(* CODESYS project l2sivacuumv1.3.3.library
   Company: SLAC - LCLS
   DefaultNamespace: LCLS_Vacuum
   Title: LCLS Vacuum
   Placeholder: LCLS Vacuum
   Author: LCLS ECS-Platforms
   Version: 1.3.3

Project tree, tasks and I/O mapping:
  libraries: LCLS General, * (SLAC); LCLSVacuumSerialDriverLib, 0.0.0 (SLAC - LCLS); PMPS, 0.12.0 (SLAC - LCLS); Tc2_DataExchange, * (Beckhoff Automation GmbH); Tc2_EtherCAT, * (Beckhoff Automation GmbH); Tc2_ModbusSrv, * (Beckhoff Automation GmbH); Tc2_Standard, * (Beckhoff Automation GmbH); Tc2_System, * (Beckhoff Automation GmbH); Tc2_TcpIp, * (Beckhoff Automation GmbH); Tc2_Utilities, * (Beckhoff Automation GmbH); Tc3_EventLogger, * (Beckhoff Automation GmbH); Tc3_JsonXml, * (Beckhoff Automation GmbH); Tc3_Module, * (Beckhoff Automation GmbH); TcUnit, * (www.tcunit.org)
  DUTs/
    Gauges/
      data type E_PressureState
      data type Gauge_Type
      data type ST_VG
    Pumps/
      data type E_PumpState
      data type ST_AgilentPTM
      data type ST_EbaraDryPump
      data type ST_EbaraEVA
      data type ST_EbaraPTM
      data type ST_KashiyamaDryPump
      data type ST_LeyboldPTM
      data type ST_PfeifferPTM
      data type ST_PIP
      data type ST_PTM
      data type ST_RoughPump
    Valves/
      data type E_ValvePositionState
      data type E_VCN
      data type E_VGC
      data type ST_ValveBase
      data type ST_VCC_NO
      data type ST_VCN
      data type ST_VFS
      data type ST_VGC
      data type ST_VGC_2S
      data type ST_VRC
      data type ST_VVC
  GVLs/
    global variables Constants
    global variables Global_Variables
  POUs/
    ADS/
      function block FB_ADS [ST]
      function block FB_ADS_WATCHDOG [ST]
      function block FB_TBOOL_ADS [ST]: ACT_Logger
    Functions/
      Deprecated/
        Gauges/
          function block FB_MKS317A [ST]: ACT_Logger, IO
          function block FB_MKS500_EP [ST]: ACT_Logger, IO, M_HVE
          function block FB_PressureState [ST]
        Valves/
          function block FB_VCC [ST]: ACT_IO, M_IsClosed, M_IsOpen, M_Set_OPN_SW
          function block FB_VCC_NO [ST]: ACT_IO, M_Close
          function block FB_VGC_AP [ST]: ACT_IO, ACT_ResetAlarms, M_IsClosed, M_IsOpen, M_Set_OPN_SW
          function block FB_VGC_EBD [ST]: ACT_IO, ACT_ResetAlarms, M_IsClosed, M_IsOpen, M_Set_OPN_SW
      Gauges/
        Interfaces/
          function block FB_Gauge_Interface [ST]
          function block FB_GaugeModbus [ST]: A_ReadMB, M_GetBit
          function block FB_TGCC_ADS [ST]: ACT_Logger
          function block FB_TGPI_ADS [ST]: ACT_Logger
        function block FB_972 [ST]: ACT_IO, M_SetBits
        function block FB_9XX [ST]: ACT_IO, ACT_Logger, M_SetBits
        function block FB_CMR362 [ST]: ACT_IO, M_SetBits
        function block FB_GaugeBase [ST]
        function block FB_GCM [ST]: ACT_IO, M_SetBits
        function block FB_ITR90 [ST]: ACT_IO, M_SetBits
        function block FB_MKS_937A [ST]: ACT_IO
        function block FB_MKS_937B [ST]: ACT_IO
        function block FB_MKS275 [ST]: ACT_Logger, IO, M_SetBits
        function block FB_MKS317 [ST]: ACT_Logger, IO
        function block FB_MKS392 [ST]: ACT_IO
        function block FB_MKS422 [ST]: ACT_Logger, IO, M_AutoOn, M_HVE
        function block FB_MKS500 [ST]: ACT_Logger, IO, M_HVE, M_SetBits
        function block FB_MKS722 [ST]: ACT_IO
        function block FB_MKS909 [ST]: ACT_IO, ACT_Logger, M_AutoOn, M_SetBits
      Pumps/
        functions/
          function F_TurboExtILK_NO [LD]
          function F_TurboExtILK_NO_1 [LD]
          function F_TurboExtILKLogic [LD]
          function F_TurboExtILKLogic_2 [LD]
          function block FB_TurboExtLogic [LD]
        Interfaces/
          function block FB_PIP_Interface_In [ST]
          function block FB_PIP_Interface_Out [ST]
          function block FB_TPIP_ADS [ST]: ACT_Logger
        function block FB_EbaraDryPump [ST]: ACT_IO, ACT_Logger
        function block FB_EbaraEVA [ST]: ACT_IO, ACT_Logger
        function block FB_KashiyamaPump [ST]: ACT_IO, M_Run
        function block FB_PIP_Gamma [ST]: ACT_IlkOverride, ACT_Logger, ACT_SetGauge, IO, M_AutoOn, M_Run
        function block FB_PTM_Agilent [ST]: ACT_Interlock, ACT_Logger, BackingPressureSetPoint, ErrorMessage, IO, M_Run, M_SetBits, M_SetCurrentScale, M_SetMaxSpeed, M_SetPowerScale, M_TurboIsOn
        function block FB_PTM_Ebara_010M [ST]: ACT_IO, ACT_Logger, BackingPressureSetPoint, M_Run
        function block FB_PTM_Ebara_011M [ST]: ACT_IO, ACT_Logger, BackingPressureSetPoint, M_Run
        function block FB_PTM_MagDriveDigital [ST]: ACT_IO, ACT_Logger, M_Run
        function block FB_PTM_Pfeiffer [ST]: ACT_IO, ACT_Logger, M_Run, M_Serial_IO
        function block FB_PTM_TurboDrive [ST]: ACT_IO, ACT_Logger, M_Run, M_Serial_IO
        function block FB_PTM_TwisTorr [ST]: ACT_IO, ACT_Logger, M_Run
        function block FB_Pump [ST]: ACT_Logger
        function block FB_ScrollPump [ST]: IO, M_Run
      Valves/
        functions/
          function F_RoughPumpInlet_ILK [ST]
          function F_TURBO_VRC_ILK [ST]
          function F_TurboGateValve_ILK [ST]
          function F_TurboGateValve_ILK_1 [ST]
          function F_TurboGateValve_Protection_ILK [ST]
          function F_VALVE_REL_ILK [ST]
          function F_VRC_DIODE_ILK [ST]
          function F_VRC_DIODE_ILK_OK [ST]
        Interfaces/
          function block FB_TVGC_2S_ADS [ST]: ACT_Logger
          function block FB_TVGC_ADS [ST]: ACT_Logger
          function block FB_Valve_Interface [ST]
          function block FB_VFS_Interface [ST]: ACT_Logger, IO
          interface ITF_Valve
        function block FB_Kashiyama_VRC [ST]: ACT_IO
        function block FB_MKS248 [ST]: ACT_IO
        function block FB_TurbVentvalve_NO [LD]: ACT_IO, M_Close
        function block FB_Valve [ST]: ACT_Logger
        function block FB_VCN [ST]: ACT_IO, M_ValveControl
        function block FB_VFS [ST]: ACT_ResetAlarms, IO
        function block FB_VGC [ST]: ACT_IO, ACT_Logger, ACT_PMPS, ACT_ResetAlarms, M_IsClosed, M_IsOpen, M_Set_OPN_SW
        function block FB_VGC_2S [ST]: ACT_IO, ACT_Logger, ACT_PMPS, ACT_ResetAlarms, M_IsClosed, M_IsOpen, M_Set_OPN_SW
        function block FB_VRC [ST]: ACT_IO, ACT_Logger, M_IsClosed, M_IsOpen, M_Set_OPN_SW
        function block FB_VRC_EBD [ST]: ACT_IO, ACT_Logger, M_IsClosed, M_IsOpen, M_Set_OPN_SW
        function block FB_VRC_NO [ST]: ACT_IO, M_IsClosed, M_IsOpen, M_Set_CLS_SW
        function block FB_VRC_OK_CLS [ST]
        function block FB_VVC [ST]: ACT_IO, M_IsClosed, M_IsOpen, M_Open, M_Set_OPN_SW
  UnitTests/
    Functions/
      function V_TO_INT [ST]
    Gauges/
      function block FB_GCC_Test [ST]: M_CheckRange, M_INIT, M_Interlock, M_SelfProtection
      function block FB_GPI_Test [ST]: M_CheckRange, M_INIT
    Pumps/
      function block FB_PIP_Test [ST]: M_AutoStart, M_Check_State, M_INIT, M_Interlock
      function block FB_PTM_Test [ST]: M_INIT, M_Interlock, M_PTM_EBARA
    Valves/
      function block FB_VGC_Test [ST]: M_Check_State, M_INIT, M_Interlock
      function block FB_VRC_Test [ST]: M_Check_State, M_INIT, M_Interlock
    program PRG_Test [ST]
  Version/
    global variables Global_Version
  VISUs/
*)

// DUTs/Gauges/E_PressureState
TYPE E_PressureState :
(
	// Invalid states
	PressInvalid,//	 //gc_GaugeValidState - 1,
	GaugeDisconnected, //gc_GaugeValidState -2,
	OoR, //gc_GaugeValidState -6,
	// Ion gauges
	Off, //gc_GaugeValidState - 3,
	Starting, //gc_GaugeValidState - 4
	
	//Valid States (Positive)
	Valid, // gc_GaugeValidState set in "Global Variable Folder: Constants"
	ValidHi, //gc_GaugeValidState + 1,
	ValidLo //gc_GaugeValidState + 2,
	
) INT;
END_TYPE

// DUTs/Gauges/Gauge_Type
TYPE Gauge_Type: ( 
PG722B := 0, //Baraton Gauge
IG903 := 1 , //Cold Cathode
PG907 := 2 , //Pirani Gauge
IG909:= 3 , //Hot Cathode
PG925 := 4 ); //MicroPirani Gauge
(* This enumeration should match up with the EDM MUX button on the vacuum gauge expert controls screen *)
END_TYPE

// DUTs/Gauges/ST_VG
TYPE ST_VG :
STRUCT
	/// A general gauge structure is used to make the rest of the interlocking simpler. There are some parameters for cold cathodes that are not used by pirani.
	///These features aren't disabled, they just aren't used, think child/parent classes. 
	/// 
	{attribute 'pytmc' := '
    pv: PRESS;
	field: HOPR 1000
	field: LOPR 0
	field: PREC 2
	field: EGU "TORR"
	io: i;
    '}
	rPRESS: REAL;  //This is the human-readable pressure
	{attribute 'pytmc' := '
    pv: AT_VAC;
	io: i;
	field: ZNAM FALSE; 
	field: ONAM TRUE;
    '}
	xAT_VAC: BOOL;
	{attribute 'pytmc' := '
    pv: PRESS_OK;
	field: ZNAM OFF; 
	field: ONAM ON;
	io: i;
    '}
	xPRESS_OK: BOOL;
	{attribute 'pytmc' := '
    pv: STATE;
	field: ZRST PressInvalid;
	field: ONST GaugeDisconnected;
	field: TWST OoR;
	field: THST Off;
	field: FRST Starting;
	field: FVST Valid;
	field: SXST ValidHi;
	field: SVST ValidLo;
	io: i;
    '}
	eState	:	E_PressureState;
	(* EPICS Controls *)	
	{attribute 'pytmc' := '
    pv: HV_SW;
	io: io;
	field: ZNAM OFF; 
	field: ONAM ON;
    '}
	xHV_SW: BOOL; // High Voltage Switch from epics
	
	/// Controls and I/Os
	{attribute 'pytmc' := '
    pv: PRESS_AI;
	io: i;
    '}
	i_iPRESS_R  :INT; // input Pressure // Link to analog Input
	{attribute 'pytmc' := '
    pv: HV_ON;
	io: i;
    '}
	i_xHV_ON	: BOOL; //  True when High Voltage is on  
	{attribute 'pytmc' := '
    pv: DISC_ACTIVE;
	field: ZNAM NO DISC; 
	field: ONAM DISC ACTIVE;
	io: i;
    '}
	i_xDisc_Active : BOOL;// Discharge Current Active 
	{attribute 'pytmc' := '
    pv: HV_DIS_DO;
	io: i;
	field: ZNAM FALSE ;
	field: ONAM TRUE ;
    '}
	q_xHV_DIS : BOOL; // Enable High Voltage when True 
	//
	wHV_RO: WORD;
		
	/// Bakeout bit 
	xBAKEOUT: BOOL;
	
	//enum for gauge type - will replace iType
	eTYPE: Gauge_Type := PG907; 
	//Gauge type, deprecated (default to pirani)
	iTYPE: INT := 2;
	// Index location of the associated Pirani Gauge
	wPG: WORD;
	
	 
	xTurnOnTime: BOOL;/// Turn on Timers for cold cathode warmup
	
	iVacSp	:	INT;/// At vacuum setpoint for all gauges
	{attribute 'pytmc' := '
    pv: VAC_SP;
	io:io;
	field: HOPR 1000
	field: LOPR 0
	field: PREC 2
	field: EGU "TORR"
	autosave_pass1: VAL DESC
    '}
	rVAC_SP: REAL := 0.001; /// At vacuum setpoint for all gauges
	/// Protection setpoint for ion gauges at which the gauge turns off, not used for pirani 
	{attribute 'pytmc' := '
    pv: PRO_SP;
	io: io;
	field: HOPR 1000
	field: LOPR 0
	field: PREC 2
	field: EGU "TORR"
	autosave_pass1: VAL DESC
    '}
	rPRO_SP: REAL := 0.001;
	{attribute 'pytmc' := '
    pv: SP_HYS;
	io: io;
	field: HOPR 1000
	field: LOPR 0
	field: PREC 2
	field: EGU "TORR"
	autosave_pass1: VAL DESC
	'}
	/// Protection setpoint hysteresis 
	rHYS_PR: REAL := 0.001; 
	{attribute 'pytmc' := '
    pv: ILK_OK;
	field: ZNAM NOT OK ;
	field: ONAM OK ;
	io: i;
	'}
	xILKOk	:	BOOL; (* also a control *)
	{attribute 'pytmc' := '
    pv: LOGGER;
	io: io;
	field: ZNAM OFF ;
	field: ONAM ON ;
    '}
	xLog : BOOL:=TRUE;
	//Required for other devices using this gauge as interlock
	sPath: STRING;

	/// Full scale pressure in Torr for baratron pressure conversion 
	rFULL_SCALE: REAL := 1000;
	
END_STRUCT
END_TYPE

// DUTs/Pumps/E_PumpState
TYPE E_PumpState :
(
pumpSTOPPED	:= 0,
pumpSTARTING	:= 1,
pumpRUNNING	:= 2,
pumpFAULT := 3,
pumpSTOPPING :=4
);
END_TYPE

// DUTs/Pumps/ST_AgilentPTM
TYPE ST_AgilentPTM EXTENDS ST_PTM :
STRUCT

(* Inputs *)
	(* 24V in Ramp state; 0V for others *)
	{attribute 'pytmc' := '
    pv: START;
	field: ZNAM FALSE; 
	field: ONAM TRUE;
	io: i;
	'}
    i_xSTART :	BOOL; 
	
	(* setpoint related to frequency *)
	{attribute 'pytmc' := '
    pv: R1Status;
	field: ZNAM FALSE; 
	field: ONAM AT SPEED;
	io: i;
	'}
	i_xR1	:  BOOL;
	
	(* setpoint related to Power *)
	{attribute 'pytmc' := '
    pv: R2Status;
	field: ZNAM FALSE; 
	field: ONAM TRUE;
	io: i;
	'}
	i_xR2	:  BOOL;
	
	(* low speed mode *)
	{attribute 'pytmc' := '
    pv: LSPD;
	field: ZNAM FALSE; 
	field: ONAM TRUE;
	io: i;
	'}
	i_xLSpd	:  BOOL;
	
	
	(* Fault input*)
	//i_xFault : BOOL;  Inherit ST_PTM.xFault
	
	

(* controls *)
	(* Start/Stop - 
		q_RunDo ;   Inherit ST_PTM.
	 *)
	
	(* Low speed control *)
	{attribute 'pytmc' := '
    pv: LSPD_DO;
	field: ZNAM FALSE; 
	field: ONAM TRUE;
	io: i;
	'}
	q_xLSpd		:  BOOL; 
	
	(*Soft start *)
	{attribute 'pytmc' := '
    pv: XSS_DO;
	field: ZNAM FALSE; 
	field: ONAM TRUE;
	io: i;
	'}
	q_xSS   	:  BOOL; 
		
	(*pump Lock*)
	{attribute 'pytmc' := '
    pv: FaultLock;
	field: ZNAM FALSE; 
	field: ONAM TRUE;
	io: i;
	'}
	xPumpFaultLock : BOOL := FALSE;
	// i_xPumpLockReset: BOOL := FALSE; Inherit ST_PTM.xReset
	// Error messages
	{attribute 'pytmc' := '
    pv: ErrorMessage;
	io: i;
	'}
	sError : STRING;
	{attribute 'pytmc' := '
	pv: Power_MON;
	io: i;
	field: PREC 2
	field: EGU "W";
	'}
	i_rPowerMon : REAL;

END_STRUCT
END_TYPE

// DUTs/Pumps/ST_EbaraDryPump
TYPE ST_EbaraDryPump EXTENDS ST_RoughPump :
STRUCT
(* Extension of the rough pump archetype for ebara 
Applicable to: 
EV-S20
EV-S50
EV-S100
EV-S200
*)

//Controls
{attribute 'pytmc' := '
    pv: MPStart;
	field: ZNAM FALSE; 
	field: ONAM TRUE;
	io: i;
    '}
q_xMPStart	:	BOOL; //Main Pump start
{attribute 'pytmc' := '
    pv: BPStart;
	field: ZNAM FALSE; 
	field: ONAM TRUE;
	io: i;
    '}
q_xBPStart	:	BOOL; // Booster Pump start (this can be started by the pump automatically)

xBPIlk	:	BOOL;	//Booster pump interlock
rBPIlkSP	:	REAL := 30; //Booster pump pressure setpoint
tonBP	:	TON := (PT:=T#5S); //Timer for pressure and valve stability


//Readbacks
{attribute 'pytmc' := '
    pv: MPStatus;
	field: ZNAM FALSE; 
	field: ONAM TRUE;
	io: i;
    '}
i_xMPStatus	:	BOOL; //MP status
{attribute 'pytmc' := '
    pv: BPStatus;
	field: ZNAM FALSE; 
	field: ONAM TRUE;
	io: i;
    '}
i_xBPStatus	:	BOOL; //BP status
{attribute 'pytmc' := '
    pv: WARN_DI;
	field: ZNAM FALSE; 
	field: ONAM TRUE;
	io: i;
    '}
i_xWarning	:	BOOL; //Warning status
{attribute 'pytmc' := '
    pv: ALARM;
	field: ZNAM FALSE; 
	field: ONAM TRUE;
	io: i;
    '}
i_xAlarm	:	BOOL; //Alarm, maps to error
{attribute 'pytmc' := '
    pv: REMOTE;
	field: ZNAM FALSE; 
	field: ONAM TRUE;
	io: i;
    '}
i_xRemote	:	BOOL; //Remote control status


END_STRUCT
END_TYPE

// DUTs/Pumps/ST_EbaraEVA
TYPE ST_EbaraEVA EXTENDS ST_RoughPump:
STRUCT

(* Output *)	
	//q_xRunDO 	:	BOOL; in Rough PUMP

	
(* Input *)
{attribute 'pytmc' := '
    pv: REMOTE;
	field: ZNAM FALSE; 
	field: ONAM TRUE;
	io: io;
    '}
	q_xRemote	:	BOOL;
	{attribute 'pytmc' := '
    pv: ALARM_OK;
	field: ZNAM FALSE; 
	field: ONAM TRUE;
	io: i
    '}
	i_xAlarmOK	:	BOOL;
	
	{attribute 'pytmc' := '
    pv: RUN_DI;
	field: ZNAM FALSE; 
	field: ONAM TRUE;
	io: i
    '}
	i_xIsRun		:	BOOL;



END_STRUCT
END_TYPE

// DUTs/Pumps/ST_EbaraPTM
TYPE ST_EbaraPTM EXTENDS ST_PTM :
STRUCT
(* Extension of the PTM archetype for Ebara turbo controllers 
Applicable to: 
ETC series
*)
//Controls
	{attribute 'pytmc' := '
    pv: START;
	field: ZNAM FALSE; 
	field: ONAM TRUE;
	io: i;
	'}
q_xStart   : BOOL; //Outputs - FB decides if these are actually set
	{attribute 'pytmc' := '
    pv: STOP;
	field: ZNAM FALSE; 
	field: ONAM TRUE;
	io: i;
	'}
q_xStop    : BOOL;
	{attribute 'pytmc' := '
    pv: RESET;
	field: ZNAM FALSE; 
	field: ONAM TRUE;
	io: i;
	'}
q_xReset   : BOOL; // xReset is momentary reset switch - resets protection functions
	{attribute 'pytmc' := '
    pv: PROT;
	field: ZNAM FALSE; 
	field: ONAM TRUE;
	io: i;
	'}
q_xProtection : BOOL; //NC. If opened, pump will decelerate/not start
	{attribute 'pytmc' := '
    pv: SETSPEED
	field: ZNAM FALSE; 
	field: ONAM TRUE;
	io: io
	'}
iq_xSpeedSet    : BOOL; //Request to set speed
	{attribute 'pytmc' := '
    pv: SPEED_REQ
	io: io
	field: EGU "Hz"
	'}
q_iSpeedSet   : DINT; //Requested speed (min. 100Hz)
	{attribute 'pytmc' := '
	pv: OVRD_ON 
	field: ZNAM OFF; 
	field: ONAM ON;
	io: io
	'}
i_xOverride   : BOOL; //Override mode - ignores interlocks

//Readbacks - also has Accel/At speed/Decel/Fault/Cur Speed (min 100RPM)
	{attribute 'pytmc' := '
    pv: ROTATE_STATUS
	field: ZNAM FALSE; 
	field: ONAM ROTATING;
	io: i
	'}
i_xRotate : BOOL; //If open, pump is rotating
	{attribute 'pytmc' := '
    pv: DECEL
	field: ZNAM FALSE; 
	field: ONAM DECELERATING;
	io: i
	'}
i_xDecel  : BOOL; //If closed, brake engaged (pump decelerating)
	{attribute 'pytmc' := '
    pv: FAULT_OK
	field: ZNAM FALSE; 
	field: ONAM TRUE;
	io: i
	'}
i_xNCFault  : BOOL; //Normally closed fault wiring. If false, there is a fault, or cable is unplugged.



END_STRUCT
END_TYPE

// DUTs/Pumps/ST_KashiyamaDryPump
TYPE ST_KashiyamaDryPump EXTENDS ST_RoughPump:
STRUCT

(* Output *)	
	//q_xRunDO 	:	BOOL; in Rough PUMP
	{attribute 'pytmc' := '
    pv: RESET_DO;
	field: ZNAM FALSE; 
	field: ONAM TRUE;
	io: i
	'}
	q_xResetDo	: 	BOOL;
	{attribute 'pytmc' := '
    pv: LSPD_DO;
	field: ZNAM FALSE; 
	field: ONAM TRUE;
	io: i
	'}
	q_xLspdDo	: 	BOOL;
	
(* Input *)
{attribute 'pytmc' := '
    pv: REMOTE;
	field: ZNAM FALSE; 
	field: ONAM TRUE;
	io: i
    '}
	i_xLocal	:	BOOL;
	{attribute 'pytmc' := '
    pv: ALARM_OK;
	field: ZNAM FALSE; 
	field: ONAM TRUE;
	io: i
    '}
	i_xAlarmOK	:	BOOL;
	{attribute 'pytmc' := '
    pv: WARN_OK;
	field: ZNAM FALSE; 
	field: ONAM TRUE;
	io: i
    '}
	i_xWarningOK	:	BOOL;
	{attribute 'pytmc' := '
    pv: RUN_DI;
	field: ZNAM FALSE; 
	field: ONAM TRUE;
	io: i
    '}
	i_xIsRun		:	BOOL;

(* Logic status *)

	xLspd_IlkENA:   BOOL;

(* EPICS *)
	//xRunSW		:	BOOL; in Rough PUMP
	{attribute 'pytmc' := '
    pv: RESET_SW;
	field: ZNAM FALSE; 
	field: ONAM TRUE;
	io: io
	'}
	xResetSW	:	BOOL; //For resetting faults
	{attribute 'pytmc' := '
    pv: LSPD_SW;
	field: ZNAM FALSE; 
	field: ONAM TRUE;
	io: io
	'}
	xLspdSW     :   BOOL;
	LowSP  :   REAL := 0.02; //Torr
	HighSP :   REAL; //Torr
    RdyTmr : REAL;
END_STRUCT
END_TYPE

// DUTs/Pumps/ST_LeyboldPTM
TYPE ST_LeyboldPTM EXTENDS ST_PTM :
STRUCT
(* Extension of the PTM archetype for Oerlikon turbo controllers 
Applicable to: 
Mag Drive Digital
Mag Drive S
More?
*)
//Readbacks
	{attribute 'pytmc' := '
    pv: DECEL;
	field: ZNAM FALSE; 
	field: ONAM TRUE;
	io: i;
	'}
	i_xDecel	:	BOOL;
	{attribute 'pytmc' := '
    pv: PWR_RBV;
	io: i;
	'}
	i_diPwr   	:   DINT;
	i_diElecTemp:	DINT;
	{attribute 'pytmc' := '
    pv: OVR_TEMP;
	field: ZNAM FALSE; 
	field: ONAM TRUE;
	io: i;
	'}
	i_xTempFault:	BOOL;
	i_xNCError	:	BOOL; //Using normally closed wiring

//Controls
	{attribute 'pytmc' := '
    pv: REMOTE;
	field: ZNAM FALSE; 
	field: ONAM TRUE;
	io: io;
	'}
	q_xRemote :BOOL;
	i_xRemote : BOOL; (* Remote control enabled *)
END_STRUCT
END_TYPE

// DUTs/Pumps/ST_PfeifferPTM
TYPE ST_PfeifferPTM EXTENDS ST_PTM :
STRUCT
(* Extension of the PTM archetype for Pfeiffer turbos 
Applicable to: 
HiPace series w/ onboard controllers
More?
*)
	{attribute 'pytmc' := '
    pv: RESET;
	field: ZNAM FALSE; 
	field: ONAM TRUE;
	io: i;
	'}
	q_xReset   : BOOL;
	//Readbacks
	{attribute 'pytmc' := '
	pv: PWR_RBV;
	io: i;
	'}
	i_diPwr		:	DINT;
	{attribute 'pytmc' := '
	pv: TempElec_RBV;
	io: i;
	'}
	i_diElecTemp	:	DINT;
	{attribute 'pytmc' := '
	pv: TempPump_RBV;
	io: i;
	'}
	i_diBtmTemp:	DINT;
	{attribute 'pytmc' := '
	pv: TempBearing_RBV;
	io: i;
	'}
	i_diBrngTemp:	DINT;
	{attribute 'pytmc' := '
	pv: TempMotor_RBV;
	io: i;
	'}
	i_diMtrTemp:	DINT;
	{attribute 'pytmc' := '
	pv: ErrorCode_RBV;
	io: i;
	'}
	i_iErrorCode	:	INT; //might change these to enumeration someday
	{attribute 'pytmc' := '
	pv: WarningCode_RBV;
	io: i;
	'}
	i_iWarningCode	:	INT;
	{attribute 'pytmc' := '
	pv: TempFault_RBV;
	field: ZNAM FALSE;
	field: ONAM TRUE;
	io: i;
	'}
	i_xTempFault	:	BOOL;
	{attribute 'pytmc' := '
	pv: Power_RBV;
	io: i;
	'}
	i_uiPowerPctRbk :   UINT;
	
	{attribute 'pytmc' := '
	pv: SET_SPEED;
	io: io;
	field: EGU "Hz"
	'}
	i_dSetSpd	:	DINT;
	
//Controls
	q_uiPowerPct : UINT := 100; //Should normally be 100
	
END_STRUCT
END_TYPE

// DUTs/Pumps/ST_PIP
TYPE ST_PIP :
STRUCT
(* Read back *)
// 	i_xHVisON : BOOL; 
	
(* Interlock *)
	{attribute 'pytmc' := '
    pv: ILK_OK;
	field: ZNAM NOT OK ;
	field: ONAM OK ;
	io: i;
	'}
   	xILKOk : BOOL; 
	
	{attribute 'pytmc' := '
    pv: ERROR;
	field: ZNAM FALSE ;
	field: ONAM TRUE ;
	io: i;
	'}
   	xError : BOOL; 
	
	{attribute 'pytmc' := '
	pv: AT_VAC_SP;
	io: io;
	field: HOPR 1000
	field: LOPR 0
	field: PREC 2
	field: EGU "TORR"
	autosave_pass1: VAL DESC
	'}
	rHVEna_SP : REAL := 1.0E-4;	
	
	{attribute 'pytmc' := '
    pv: ILK_DEVICE;
	io: i;
    '}
	sIlkDeviceName: STRING;
	//Required for other devices using this gauge as interlock
	sPath: STRING;
	
(* EPICS Controls *)	
	{attribute 'pytmc' := '
    pv: HV_SW;
	io: io;
	field: ZNAM OFF; 
	field: ONAM ON;
    '}
	xHVEna_SW : BOOL; 
	{attribute 'pytmc' := '
    pv: Auto_On;
	field: ZNAM FALSE; 
	field: ONAM TRUE;
	io:i;
    '}
	xAutoOn : BOOL;

	{attribute 'pytmc' := '
	pv: OVRD_ON ;
	field: ZNAM Override OFF ;
	field: ONAM Override ON;
	io: io;
	'}
	xOverrideMode	:	BOOL; (* Shows the override status of this valve *)
	
	{attribute 'pytmc' := '
    pv: FORCE_START;
	io: io;
	field: ZNAM FALSE;
	field: ONAM FORCE START;
    '}
	pv_xOvrdStart	:	BOOL;
	

	{attribute 'pytmc' := '
    pv: SP_HYS;
	io: io;
	field: HOPR 1000
	field: LOPR 0
	field: PREC 2
	field: EGU "TORR"
	autosave_pass1: VAL DESC
	'}
	/// Protection setpoint hysteresis 
	rHYS_PR: REAL := 0.001; 
	{attribute 'pytmc' := '
    pv: AI_Offset;
	io: io;
    '}
	iOffset: INT:=13;
	{attribute 'pytmc' := '
    pv: Inverted;
	field: ZNAM NORMAL; 
	field: ONAM INVERTED;
	io: io;
    '}
	bOutputInverted : BOOL;
(* IO Controls *)
	{attribute 'pytmc' := '
    pv: HV_DO;
	field: ZNAM OFF; 
	field: ONAM ON;
	io: i;
    '}
	q_xHVEna_DO : BOOL;	// Enable High Voltage when True // 'TcLinkTo' (EL1124) ^Input
	{attribute 'pytmc' := '
    pv: PRESS;
	field: HOPR 1000
	field: LOPR 0
	field: PREC 2
	field: EGU "TORR"
	io: i;
    '}
	rPRESS: REAL;  //
	{attribute 'pytmc' := '
    pv: PRESS_AI;
	io: i;
    '}
	i_iPRESS: REAL;  //
	{attribute 'pytmc' := '
    pv: HV_DI;
	field: ZNAM FALSE; 
	field: ONAM TRUE;
	io:i;
    '}
	i_xHV_DI : BOOL; // NO contact // 'TcLinkTo' (EL1004) ^Input

	{attribute 'pytmc' := '
	pv: STATE;
	field: ZRST STOPPED;
	field: ONST STARTING;
	field: TWST RUNNING;
	field: THST FAULT;
	field: FRST STOPPING;
	io: i;
	'}

	eState	:	E_PumpState;
	
	{attribute 'pytmc' := '
    pv: LOGGER;
	io: io;
	field: ZNAM OFF ;
	field: ONAM ON ;
    '}
	xLog : BOOL:=TRUE;
END_STRUCT
END_TYPE

// DUTs/Pumps/ST_PTM
TYPE ST_PTM :
STRUCT
(* General PTM Structure
Each PTM might have a serial control structure, but all will have a general supervisory control structure

NOTE: This is an archetype, use an extension of this structure for a specific pump (or make one).

*)

(* Controls *)
	{attribute 'pytmc' := '
	pv: RUN_SW;
	field: ZNAM STOP; 
	field: ONAM RUN;
	io: io;
	'}
	xRunSW	:	BOOL;
	{attribute 'pytmc' := '
	pv: RST_SW;
	field: ZNAM FALSE; 
	field: ONAM TRUE;
	io: io;
	'}
	xResetSW	:	BOOL; //For resetting faults
	{attribute 'pytmc' := '
    pv: RUN_DO;
	io: i;
	'}
	q_RunDO 	:	BOOL;

(* Readbacks *)
    {attribute 'pytmc' := '
	pv: ILK_OK;
	field: ZNAM ILK ACTIVE;
	field: ONAM ILK OK;
	io: i;
	'}
	xExtRunOk	:	BOOL; (* also a control *)
	{attribute 'pytmc' := '
    pv: ACCEL;
	field: ZNAM FALSE; 
	field: ONAM TRUE;
	io: i;
	'}
	i_xAccel	:	BOOL;
	{attribute 'pytmc' := '
    pv: AT_SPD;
	field: ZNAM FALSE; 
	field: ONAM AT SPEED;
	io: i;
	'}
	i_xAtSpd	:	BOOL;
	{attribute 'pytmc' := '
	pv: SPEED;
	io: i;
	field: EGU "Hz"
	'}
	i_diCurSpd	:	DINT;
	
	xCommTimeout	:	BOOL := TRUE;  (* Initialized true since we haven't talked to pump yet *)
(* Alarm Outputs *)
	{attribute 'pytmc' := '
    pv: FAULT;
	field: ZNAM FALSE; 
	field: ONAM TRUE;
	io: i;
	'}
	i_xFault		:	BOOL; (*FAULT*)
	{attribute 'pytmc' := '
    pv: WARN;
	field: ZNAM FALSE; 
	field: ONAM TRUE;
	io: i;
	'}
	i_xWarn		:	BOOL; (* warning *)
	{attribute 'pytmc' := '
    pv: ALARM;
	field: ZNAM FALSE; 
	field: ONAM TRUE;
	io: i;
	'}
	i_xALARM	:	BOOL; (* ALARM *)
	
(* IWS instructions *)
	xActive	:	BOOL; // this bit is set to add the pump to the system
	iPumpGrp 	:	INT; // all members of a pump group start at the same time
	
(* Operational Setpoints *)
	rForelineSP	:	REAL := 0.5;
	
	{attribute 'pytmc' := '
    pv: BP_SP;
	io: io;
	field: HOPR 1000
	field: LOPR 0
	field: PREC 2
	field: EGU "TORR"
	autosave_pass1: VAL DESC
	'}
	rBackingPressureSP : REAL := 0.01;
	{attribute 'pytmc' := '
    pv: IP_SP;
	io: io;
	field: HOPR 1000
	field: LOPR 0
	field: PREC 2
	field: EGU "TORR"
	autosave_pass1: VAL DESC
	'}
	rInletPressureSP : REAL := 0.02; //20mTorr
(*State*)	
	{attribute 'pytmc' := '
	pv: STATE;
	field: ZRST STOPPED;
	field: ONST STARTING;
	field: TWST RUNNING;
	field: THST FAULT;
	field: FRST STOPPING;
	io: i;
	'}

	eState	:	E_PumpState;
	
	{attribute 'pytmc' := '
	pv: CURR_MON;
	io: i;
	field: PREC 2
	field: EGU "A";
	'}
	i_rCurrentMon : REAL;

	{attribute 'pytmc' := '
    pv: TEMP_MON;
	io: i;
	field: PREC 2;
	field: EGU "C";
	'}
	i_rTempMon	:	REAL;
 
	{attribute 'pytmc' := '
    pv: LOGGER;
	io: i;
	field: ZNAM OFF ;
	field: ONAM ON ;
    '}
	xLog : BOOL:=TRUE;


END_STRUCT
END_TYPE

// DUTs/Pumps/ST_RoughPump
TYPE ST_RoughPump :
STRUCT
	
(* Generic roughing pump controls 

NOTE: This is an archetype, use an extension of this structure for a specific pump (or make one).

*)

//Controls
{attribute 'pytmc' := '
    pv: RUN_SW;
	field: ZNAM Stop; 
	field: ONAM Start;
	io: io;
	'}
pv_xRunSW	:	BOOL; //epics/ software control switch
{attribute 'pytmc' := '
    pv: RUN_DO;
	field: ZNAM FALSE; 
	field: ONAM TRUE;
	io: i
	'}
q_xRunDo 	:   BOOL; 

//Status and Readback
{attribute 'pytmc' := '
    pv: ILK_OK;
	field: ZNAM NOT OK ;
	field: ONAM OK ;
	io: i
	'}
xIlkOK	:	BOOL; //Interlock bit, true means OK to run
xExtIlk	:	BOOL; //External interlock, this is where the logic goes
{attribute 'pytmc' := '
    pv: AT_SPD;
	field: ZNAM FALSE; 
	field: ONAM TRUE;
	io: i
	'}
xAtSpd	:	BOOL; //Pump at speed setpoint
{attribute 'pytmc' := '
    pv: WARN;
	field: ZNAM FALSE; 
	field: ONAM TRUE;
	io: i
	'}
xWrn	:	BOOL; //Pump warning
iWrn	:	BOOL; //Warning state/code
{attribute 'pytmc' := '
    pv: ERROR;
	field: ZNAM FALSE; 
	field: ONAM TRUE;
	io: i
	'}
xErr	:	BOOL; //Error summary
iErr	:	BOOL; //Error state/code

(*State*)	
	{attribute 'pytmc' := '
	pv: STATE;
	field: ZRST STOPPED;
	field: ONST STARTING;
	field: TWST RUNNING;
	field: THST FAULT;
	field: FRST STOPPING;
	io: i;
	'}

	eState	:	E_PumpState;

END_STRUCT
END_TYPE

// DUTs/Valves/E_ValvePositionState
TYPE E_ValvePositionState :
	(
OPEN	:= 0,
CLOSED	:= 1,
MOVING	:= 2,
INVALID :=3,
OPEN_F :=4
);
END_TYPE

// DUTs/Valves/E_VCN
TYPE E_VCN :
	(
CloseValve	:= 0,
OpenValve	:= 1,
PressureControl	:= 2,
ManualControl	:= 3

	);
END_TYPE

// DUTs/Valves/E_VGC
TYPE E_VGC :
(

	Vented,
	AtVacuum,
	ERR_DiffPress,
	ERR_LostVac,
	ERR_ExtFault,
	At_Vac,
	Triggered,
	Vac_Fault,
	Cls_Timeout,
	Opn_Timeout


);
END_TYPE

// DUTs/Valves/ST_ValveBase
TYPE ST_ValveBase :
STRUCT
	(* EPICS Controls *)
	{attribute 'pytmc' := '
	pv: OPN_SW; 
	field: ZNAM CLOSE; 
	field: ONAM OPEN;
	io: io ;
	'}
	pv_xOPN_SW	: BOOL;
	{attribute 'pytmc' := '
    pv: ALM_RST;
	io: io;
    '}
	pv_xAlmRst	: BOOL;
	{attribute 'pytmc' := '
    pv: FORCE_OPN;
	io: io;
	field: ZNAM FALSE;
	field: ONAM FORCE OPEN;
    '}
	pv_xOvrdOpn	:	BOOL;

	{attribute 'pytmc' := '
	pv: OVRD_ON ;
	field: ZNAM Override OFF ;
	field: ONAM Override ON;
	io: io;
	'}
	xOverrideMode	:	BOOL; (* Shows the override status of this valve *)

(* I/Os*)
(* Readbacks *)
	{attribute 'pytmc' := '
	pv: OPN_DI;
	io: i;
	field: ZNAM FALSE;
	field: ONAM OPEN;
	'}
	i_xOpnLS	: BOOL;
	{attribute 'pytmc' := '
    pv: CLS_DI;
	io: i;
	field: ZNAM FALSE;
	field: ONAM CLOSE;
    '}
	i_xClsLS	: BOOL;
(* Controls *)
	{attribute 'pytmc' := '
    pv: OPN_DO;
	io: i;
	field: ZNAM FALSE;
	field: ONAM TRUE;
    '}
	q_xOPN_DO	: BOOL;
(* Interlocks *)
	{attribute 'pytmc' := '
	pv: EXT_ILK_OK ;
	field: ZNAM NOT OK ;
	field: ONAM OK ;
	io: i ;
	'}
	xEXT_OK	:	BOOL := FALSE;	(* External interlock for custom interlocking in addition to regular DP ilk, this must be set true, or the interlock condition before calling the FB_VGC *)

	
	{attribute 'pytmc' := '
    pv: OPN_OK;
	field: ZNAM OPN ILK NOT OK ;
	field: ONAM OPN ILK OK ;
	io: i;
 	'}
	xOPN_OK	:	BOOL;	(* Final SUM of DP_OK and EXT_OK, needed because it allows the DP ilk to be switched off, see FB_VGC.Dis_DPIlk *)
	
(* States *)	
{attribute 'pytmc' := '
	pv: POS_STATE;
	type: mbbi ;
	field: ZRST OPEN ;
	field: ONST CLOSED ;
	field: TWST MOVING ;
	field: THST INVALID ;
	field: FRST OPEN_F ;
	io: i;
	'}
	eState	:	E_ValvePositionState := INVALID;

	{attribute 'pytmc' := '
	pv: STATE;
	field: ZRST Vented;
	field: ONST At Vacuum;
	field: TWST Differential Pressure;
	field: THST Lost Vacuum;
	field: FRST Ext Fault;
	field: FVST AT Vacuum;
	field: SXST Triggered;
	field: SVST Vacuum Fault;
	field: EIST Close Timeout;
	field: NIST Open Timeout;
	io: i;
	'}
	eVGC_State : E_VGC;

(* Error *)
	
	{attribute 'pytmc' := '
    pv: ERROR;
	field: ZNAM NO ERROR ;
	field: ONAM ERROR PRESENT ;
	io: o;
    '}
	bErrorPresent : BOOL;
	iErrorCode: INT;
	{attribute 'pytmc' := '
    pv: ErrMsg;
	io: o;
    '}
	sErrorMessage: STRING;
	{attribute 'pytmc' := '
    pv: LOGGER;
	io: io;
	field: ZNAM OFF ;
	field: ONAM ON ;
    '}
	xLog : BOOL:=TRUE;

END_STRUCT
END_TYPE

// DUTs/Valves/ST_VCC_NO
TYPE ST_VCC_NO:
STRUCT

(* A normally open valve needs permission to close! *)
(* Inputs *)
	{attribute 'pytmc' := '
	pv: CLS_SW ;
	field: ONAM CLOSE; 
	field: ZNAM OPEN;
	io: io ;
	'}
	pv_xCLS_SW	: BOOL;
	{attribute 'pytmc' := '
    pv: FORCE_CLS;
	field: ZNAM FALSE;
	field: ONAM FORCE CLOSE;
	io: io;
	'}
	pv_xOvrdCls	:	BOOL;
	{attribute 'pytmc' := '
    pv: CLS_OK;
	field: ZNAM FALSE; 
	field: ONAM CLS_OK;
	io: i;
	'}
	xCLS_OK	: BOOL;
	
	{attribute 'pytmc' := '
	pv: OVRD_ON;
	field: ZNAM Override OFF ;
	field: ONAM Override ON;
	io: io
	'}
	xOverrideMode	:	BOOL; (* Shows the override status of this valve *)

(* Outputs *)
	{attribute 'pytmc' := '
    pv: CLS_DO;
		field: ZNAM FALSE; 
	field: ONAM TRUE;
	io: i;
	'}
	xCLS_DO	: BOOL;

END_STRUCT
END_TYPE

// DUTs/Valves/ST_VCN
TYPE ST_VCN :
STRUCT
	(* VCN - Valve Controlled Needle
	Used for Pfeiffer EVR 116 needle valves *)
	{attribute 'pytmc' := '
	pv: OPN_SW; 
	field: ZNAM CLOSE; 
	field: ONAM OPEN;
	io: io ;
	'}
	xOPN_SW	: BOOL;
	{attribute 'pytmc' := '
    pv: POS_RDBK;
	io: i;
    '}
	// Inputs
	i_iPosition	:	REAL; //Position readback (if it exists)
	
	// Outputs
	{attribute 'pytmc' := '
	pv: POS_AO_R;
	io: i ;
	'}
	q_iRawPosition	:	INT; //Position control 
	//For the EVR 116 this is 0-10V analog 0.4 closed to 9.1 Closed
	
	//Softvariables
	{attribute 'pytmc' := '
    pv: ILK_OK;
	field: ZNAM NOT OK ;
	field: ONAM OK ;
	io: i;
    '}
	xIlkOK	:	BOOL := FALSE; // Interlock Bit
	
	rUpperLimit	:	REAL:=100; // Percentage9.1;	//Upper limit on valve open
	{attribute 'pytmc' := '
	pv: POS_REQ;
	io: io;
	'}
	rReqPosition	:	REAL; //Requested position (0.0-100.0%)
	{attribute 'pytmc' :=  ' 
	pv: STATE ;
	field: ZRST Close ;
	field: ONST Open;
	field: TWST PressureControl ;
	field: THST ManualControl ;
	io: io
	'}
	eValveControl	:	E_VCN := CloseValve; // Valve control state

	ftIlk	:	F_TRIG;	

END_STRUCT
END_TYPE

// DUTs/Valves/ST_VFS
TYPE ST_VFS EXTENDS ST_ValveBase:
STRUCT

(* Interlock *)
	{attribute 'pytmc' := '
	pv: TRIG; 
	field: ZNAM TRIG_OFF; 
	field: ONAM TRIG_ON;
	io: i ;
	'}
	i_xTrigger : BOOL;
(* Commands *)
	{attribute 'pytmc' := '
	pv: CLS_SW; 
	field: ZNAM FALSE; 
	field: ONAM CLOSE;
	io: io ;
	'}
	xCLS_SW AT%Q*:BOOL; (*external open signal e.g epics*)
	
(* Alarm Outputs *)
	{attribute 'pytmc' := '
    pv: ERR_Ext;
	field: ZNAM NO ERROR ;
	field: ONAM External error present ;
	io: i;
    '}
	xERR_ExtFault		: 	BOOL;
	{attribute 'pytmc' := '
	pv: VAC_FAULT_OK; 
	field: ZNAM FAULT ; 
	field: ONAM FAULT OK;
	io: i ;
	'}
	i_xVAC_FAULT_OK : BOOL; (*Valve Vacuum OK, is set to False when there is Vacuum Fault*)

	
(*ILK Devices*)
	{attribute 'pytmc' := '
    pv: GFS;
	io: i;
    '}	
	sGFS: String;

END_STRUCT
END_TYPE

// DUTs/Valves/ST_VGC
TYPE ST_VGC EXTENDS ST_ValveBase:
STRUCT

	
(* Interlocks *)

	{attribute 'pytmc' := '
    pv: DP_OK;
	field: ZNAM DP NOT OK ;
	field: ONAM DP OK ;
	io: i;
    '}
	xDP_OK	:	BOOL;	(* Managed by the VGC function (FB_VGC) *)// Indicates the valve can be opened because the differential pressure is low enough

	{attribute 'pytmc' := ' 
	pv: AT_VAC_SP;
	io: o;
	field: HOPR 1000
	field: LOPR 0
	field: PREC 2
	field: EGU "TORR"
	autosave_pass1: VAL DESC
	'}
	rAT_VAC_SP	:	REAL := 0.000001;	// Interlock setpoint for gauges on both sides of valve
	rAT_VAC_SP_LAST	:	REAL :=0.000001 ;	// Interlock setpoint for gauges on both sides of valve
	{attribute 'pytmc' := '
    pv: AT_VAC_HYS;
	io: o;
	field: HOPR 1000
	field: LOPR 0
	field: PREC 2
	field: EGU "TORR"
	autosave_pass1: VAL DESC
    '}
	rAT_VAC_HYS	:	REAL :=0.000001;	// Hysteresis of the vacuum sp
	{attribute 'pytmc' := '
    pv: HYST_PERC ;
	io: o;
	autosave_pass1: VAL DESC
    '}
	rHYST_PERC	:	REAL := 0.80;	// Hysteresis percentage

	{attribute 'pytmc' := '
	pv: AT_VAC ; 
	field: ZNAM NOT AT VAC ;
	field: ONAM AT VAC ;
	io: i;
	'}
	xAT_VAC	:	BOOL;	//At vacuum setpoint


(* Alarm Outputs *)
	{attribute 'pytmc' := '
    pv: ERR_DifPres;
	field: ZNAM NO ERROR ;
	field: ONAM Diffrential error present ;
	io: i;
    '}
	xERR_DifPres		: 	BOOL;
	{attribute 'pytmc' := '
    pv: ERR_SP;
	field: ZNAM NO ERROR ;
	field: ONAM Setpoint error present ;
	io: i;
    '}
	xERR_SP			: 	BOOL;
	{attribute 'pytmc' := '
    pv: ERR_Ext;
	field: ZNAM NO ERROR ;
	field: ONAM External error present ;
	io: i;
    '}
	xERR_ExtFault		: 	BOOL;
	xAlmSum			: 	BOOL;
	
(*ILK Devices*)
{attribute 'pytmc' := '
    pv: ILK_DEVICE_US;
	io: i;
    '}
	sIlkUSDeviceName: STRING;
	{attribute 'pytmc' := '
    pv: ILK_DEVICE_DS;
	io: i;
    '}
	sIlkDSDeviceName: STRING;

END_STRUCT
END_TYPE

// DUTs/Valves/ST_VGC_2S
TYPE ST_VGC_2S EXTENDS ST_VGC:
STRUCT
	{attribute 'pytmc' := ' 
	pv: AT_VAC_SP_DS;
	io: o;
	field: HOPR 1000
	field: LOPR 0
	field: PREC 2
	field: EGU "TORR"
	autosave_pass1: VAL DESC
	'}
	rAT_VAC_SP_DS	:	REAL := 0.000001;	// Interlock setpoint for gauges on the downstream side of the valve
	{attribute 'pytmc' := '
    pv: AT_VAC_HYS_DS;
	io: o;
	field: HOPR 1000
	field: LOPR 0
	field: PREC 2
	field: EGU "TORR"
	autosave_pass1: VAL DESC
    '}
	rAT_VAC_HYS_DS	:	REAL :=0.000001;	// Hysteresis of the vacuum sp downstream
	rAT_VAC_SP_LAST_DS :	REAL :=0.000001 ;
END_STRUCT
END_TYPE

// DUTs/Valves/ST_VRC
TYPE ST_VRC EXTENDS ST_ValveBase:
STRUCT
(* Readbacks *)
	//In case VRC is normally open
	{attribute 'pytmc' := '
    pv: CLS_OK;
	io: i;
    '}
	xCLS_OK : BOOL := TRUE;

END_STRUCT
END_TYPE

// DUTs/Valves/ST_VVC
TYPE ST_VVC :
STRUCT

(* Inputs *)

	{attribute 'pytmc' := '
	pv: OPN_SW;
	field: ZNAM CLOSE;
	field: ONAM OPEN;
	io: io;
	'}
	pv_xOPN_SW	: BOOL;
	{attribute 'pytmc' := '
	pv:FORCE_OPN;
	field: ZNAM FALSE;
	field: ONAM OPEN;
	io: io;
	'}
	xOvrdOpn	:	BOOL;
	{attribute 'pytmc' := '
	pv: OVRD_ON;
	field: ZNAM Override ON ;
	field: ONAM Override OFF;
	io: io;
	'}
	xOverrideMode	:	BOOL; (* Shows the override status of this valve *)
	{attribute 'pytmc' := '
    pv: OPN_OK;
	field: ZNAM OPN ILK NOT OK ;
	field: ONAM OPN ILK OK ;
	io: i;
	'}
	xOPN_OK	: BOOL;

(* Outputs *)
	{attribute 'pytmc' := '
	pv: OPN_DO;
	field: ZNAM CLOSE;
	field: ONAM OPEN;
	io: i;
	'}
	q_xOPN_DO	: BOOL;

END_STRUCT
END_TYPE

// GVLs/Constants
VAR_GLOBAL CONSTANT
	gc_iSizeOfGGOArray : INT := 50;
	gc_GaugeValidState :	INT := 4;
END_VAR

// GVLs/Global_Variables
VAR_GLOBAL
	g_iSizeOfGGOArray : INT := 50;
	
	g_stSystem	:	ST_System(*System_Struct*):= (
    	xFirstScan := TRUE
	);
	
	g_DummyVG	:	ST_VG;
	
	
	 fbGetCurTaskIdx : GETCURTASKINDEX;
	 


END_VAR

// Version/Global_Version
{attribute 'TcGenerated'}
// This function has been automatically generated from the project information.
VAR_GLOBAL CONSTANT
	{attribute 'const_non_replaced'}
	{attribute 'linkalways'}
	stLibVersion_LCLS_Vacuum : ST_LibVersion := (iMajor := 1, iMinor := 3, iBuild := 3, iRevision := 0, sVersion := '1.3.3');
END_VAR

// POUs/ADS/FB_ADS
FUNCTION_BLOCK FB_ADS
VAR_INPUT
END_VAR
VAR_OUTPUT
END_VAR
VAR
	 fbLogger : FB_LogMessage := (eSubsystem:=E_SubSystem.FIELDBUS);
	tErrorPresent : R_TRIG;
END_VAR

END_FUNCTION_BLOCK

// POUs/ADS/FB_ADS_WATCHDOG
(*This function block is to be used whenever deivce data going to be read over ADS*)
(*The remote plc has to instantiate this function block in order to write a watchdog variable*)
(*that the ADS read function expects to keep checking*)
FUNCTION_BLOCK FB_ADS_WATCHDOG
VAR_INPUT
	sNetId : String; //NetID of the Destination PLC controller
	nPort : uint; // port number
	sVarName : string;// the variable name of the watchdog on the remote plc.
END_VAR
VAR_OUTPUT
	bError:BOOL;
END_VAR
VAR
	
	fb_WriteWatchdog:FB_WriteWatchdog;
	ftReset_Watchdog: F_TRIG;
	xFirstPass: BOOL:= true;
	
END_VAR



ftReset_Watchdog(CLK:= fb_WriteWatchdog.bBusy OR xFirstPass);
xFirstPass := false;

(*calling ADS Watchdog function*)
fb_WriteWatchdog(
	bEnable:= TRUE , 
	sNetId:= sNetId, 
	nPort:= nPort, 
	nIdxGrp:= , 
	nIdxOffs:= , 
	sVarName:= sVarName, 
	tWatchdogTime:= t#30ms, 
	bSendNow:= ftReset_Watchdog.Q , 
	bBusy=> , 
	nLastCnt=>  , 
	bError=> bError, 
	nErrorId=> );

	
(*Error*)

END_FUNCTION_BLOCK

// POUs/ADS/FB_TBOOL_ADS
(* This function block is created for interface a boolean singal between different PLCs*)
(* The variable values are read via ADS using the symbol name*)
FUNCTION_BLOCK FB_TBOOL_ADS Extends FB_ADS
VAR_INPUT
	sNetId : String; //NetID of the Destination PLC controller
	nPort : uint; // port number
	sVarName : string;// the variable name of the declared pip/pin function block.
	iWatchdog:UDINT;//The watchdog variable name written to by the remote plc
END_VAR
VAR_OUTPUT
	{attribute 'pytmc' := 'pv: value'}
	bBool : BOOL;
	{attribute 'pytmc' := 'pv: error'}
	bError: BOOL;
END_VAR
VAR
	fb_CheckWatchdog: FB_CheckWatchdog;
	fb_Read: FB_ReadAdsSymByName;
	ftReset: F_TRIG;
	xFirstPass: BOOL:= true;
	
END_VAR


ftReset(CLK:= fb_Read.bBusy OR xFirstPass);
xFirstPass := false;
(*calling ADS read function*)
	
fb_Read(
	bRead:=ftReset.Q , 
	sNetId:= sNetId, 
	nPort:= nPort, 
	sVarName:= sVarName, 
	nDestAddr:= ADR(bBool), 
	nLen:= SIZEOF(bBool), 
	tTimeout:= , 
	eComMode:=eAdsComModeFastCom , 
	bBusy=> , 
	bError=> , 
	nErrorId=> );	
	

(*Error*)
fb_CheckWatchdog(
	bEnable:= TRUE, 
	tWatchdogTime:= T#900ms, 
	nCnt:= iWatchdog , 
	bWatchdog=> , 
	nLastCnt=> );

bError:= fb_Read.bError OR fb_CheckWatchdog.bWatchdog;
tErrorPresent(CLK:=bError);

IF (fb_Read.bError OR fb_CheckWatchdog.bWatchdog) THEN
	bBool := FALSE; // If there is an error in connection the signal turns to FALSE
END_IF;

(*Logger*)
ACT_Logger();

ACTION ACT_Logger:
IF tErrorPresent.Q THEN
 IF(fb_Read.bError) THEN fbLogger(sMsg:='ADS Read Error', eSevr:=TcEventSeverity.Critical); END_IF;
 IF(fb_CheckWatchdog.bWatchdog) THEN fbLogger(sMsg:='ADS Watchdog Error', eSevr:=TcEventSeverity.Critical); END_IF;
END_IF
END_ACTION

END_FUNCTION_BLOCK

// POUs/Functions/Deprecated/Gauges/FB_MKS317A
(*Deprecated*)
(* This function is for the Pirani MKS 317 connected to a 937A*)
(* This function block is used to provide protection and automatic turn on of ion gauges,
 it also manages the turn on of the AT_VAC boolean, and checks to make sure the pressure is good *)
{attribute 'obsolete' := 'FB_MKS317A has been deprecated and is not valid!'} 
FUNCTION_BLOCK FB_MKS317A  Extends FB_GaugeBase
VAR_IN_OUT
	
END_VAR
VAR_INPUT
	
END_VAR
VAR_OUTPUT
	{attribute 'pytmc' := '
    pv: 
	'}
	PG : ST_VG;
END_VAR
VAR
	rV	:	REAL;
	rMinPressure: REAL := 1E-3;
	rDefaultVAC_SP: REAL :=5E-2; // Default 50 mT
	rValidLoBoundary	:	REAL := 0.2;//Manual page 61
	rValidHiBoundary	:	REAL := 9.7; //manual oage 61
	rDisconnectedBoundary	:	REAL := 0.17;
	rNoSensorBoundary	:	REAL := 10;
	(*IO*)
	i_iPRESS_R AT%I* :INT; // input Pressure // Link to analog Input
END_VAR

(* 937B Logarithmic Output Conversion *)
(* 5-20-2016, Alex Wallace and Scott Stubbs *)
(* 09-28-2018, Margaret Ghaly *)
(* This function will read the pressure from any gauge on a 937A. *)

rV := 10*INT_TO_REAL(PG.i_iPRESS_R)/32767;
PG.rPRESS := LREAL_TO_REAL(EXPT(10,((rV)/0.6)-12)); //manual page 61 937A


//Default setpoint 
IF PG.rVAC_SP = 0 THEN
	PG.rVAC_SP := rDefaultVAC_SP;
END_IF

IF (rV <=9.7 ) AND (rV>=0.6) THEN
	PG.eState := Valid; // normal
ELSIF rV >= 0.18 AND rV <= 0.22 THEN
	PG.eState := ValidLo; //LO
	PG.rPRESS := rMinPressure;
ELSIF rV > 9.7 AND rV<= 9.9 THEN
	PG.eState := ValidHi; //HIGH
ELSIF rV < 0.18 THEN
	PG.eState := GaugeDisconnected; //not on
	PG.rPRESS := -1;
ELSE
	PG.eState := PressInvalid; //other fault - could be no gauge, controller powering up etc
	PG.rPRESS := -1;
END_IF

(* Pressure OK check *)
(* Pressure gauge OK checks *)
PG.xPRESS_OK := (rV <=rValidHiBoundary ) AND (rV>=rDisconnectedBoundary);
//PG.xPRESS_OK := (PG.rPRESS >= rMinPressure);

(* Setpoint evaluation *)
PG.xAT_VAC := (*(PG.eState =Valid)*) PG.xPRESS_OK AND PG.rPRESS <= PG.rVAC_SP;

(*Logger*)
ACT_Logger();
(*soft io*)
IO();

ACTION ACT_Logger:
IF (PG.xLog) THEN
//STATE Logger  
IF ePrevState <> PG.eState THEN
	  CASE PG.eState OF
		ValidHi:
			fbLogger(sMsg:='Gauge pressure valid high.', eSevr:=TcEventSeverity.Info);
		ValidLo:
			fbLogger(sMsg:='Gauge pressure valid low.', eSevr:=TcEventSeverity.Info);
		Valid:
			fbLogger(sMsg:='Gauge pressure valid.', eSevr:=TcEventSeverity.Info);
  		GaugeDisconnected:
			fbLogger(sMsg:='Gauge Disconnected.', eSevr:=TcEventSeverity.Critical);
		PressInvalid:
			fbLogger(sMsg:='Gauge pressure invalid.', eSevr:=TcEventSeverity.Warning);
		OoR:
			fbLogger(sMsg:='Gauge pressure out of range.', eSevr:=TcEventSeverity.Warning);
		Starting:
			fbLogger(sMsg:='Gauge starting.', eSevr:=TcEventSeverity.Info);
	  END_CASE
	  ePrevState := PG.eState;  
  END_IF
 END_IF
END_ACTION

ACTION IO:
PG.i_iPRESS_R :=i_iPRESS_R;
PG.sPath := sPath;
END_ACTION

END_FUNCTION_BLOCK

// POUs/Functions/Gauges/FB_GaugeBase
{attribute 'reflection'} 
FUNCTION_BLOCK FB_GaugeBase
VAR_INPUT
END_VAR
VAR_OUTPUT
	
END_VAR
VAR
	//Logging 
    fbLogger : FB_LogMessage := (eSubsystem:=E_SubSystem.VACUUM);
    ePrevState : E_PressureState;
    tErrorPresent : R_TRIG;
    tAction : R_TRIG; // Primary action of this device (OPN_DO, etc.)
    tOverrideActivated : R_TRIG;
	 tState : R_TRIG;
	{attribute 'instance-path'}
	{attribute 'noinit'}
	sPath: STRING;
END_VAR

END_FUNCTION_BLOCK

// POUs/Functions/Deprecated/Gauges/FB_MKS500_EP
(*Deprecated*)
(* This function is for the Cold Cathode MKS 500 connected to Beckhoff EP boxes.
A separate function block is necessary for the MKS500-to-EP box interface beacuse the EP
boxes do not natively support the 5v IO signals on the MKS500 gauge.*)
(*This function provides ILK and Set Point Protection for the Cold Cathode*)
(* 500 Logarithmic Output Conversion, factory default configuration *)
{attribute 'obsolete' := 'FB_MKS500_EP has been deprecated and is not valid!'}
FUNCTION_BLOCK FB_MKS500_EP EXTENDS FB_GaugeBase
VAR_IN_OUT
		
END_VAR
VAR_INPUT
	
	PG	:	ST_VG;
END_VAR
VAR_OUTPUT
{attribute 'pytmc' := '
    pv: 
	'}
	IG : ST_VG;
END_VAR
VAR
	rV : REAL;
	GaugeTurnOnTmr : TON;

	(*IOs to be linked*)
	/// Controls and I/Os
	i_iPRESS_R AT %I* :INT; // input Pressure // Link to analog Input
	q_xHV_DIS AT %Q* : BOOL; // Enable High Voltage when True // 'TcLinkTo' (EP2624) ^Output
	//
END_VAR

VAR CONSTANT
	// Ranges has to match the configurator software
	pBase : REAL :=1.0E-10;//default curve base pressure is 1E-10. Confusing since can't actually read that low using analog out.
	vBase : REAL := 1;
	vDisconnected : REAL:= 0.5;
	vSlope : REAL := 1.0; 
	vGaugeOff: REAL := 9.8;
	vNoDischarge: REAL := 9.3;
	MinPressure: REAL := 1E-10;
	cDefaultPressure : REAL := 0;
END_VAR

(* 500 Logarithmic Output Conversion, factory default configuration *)
{attribute 'obsolete' := 'FB_VCC_NO has been deprecated and is not valid!'}
rV := 10*INT_TO_REAL(IG.i_iPRESS_R)/32767;

(* Set Guage State based on the Analog voltage*)
IF rV < vDisconnected THEN
	IG.eState := GaugeDisconnected;
	IG.rPRESS := cDefaultPressure;
ELSIF rV >= vDisconnected AND rV < (vNoDischarge -0.3)  THEN
	IG.eState := Valid;
	IG.rPRESS := LREAL_TO_REAL(EXPT(10,((rV-vBase)/vSlope+LOG(pBase))));
ELSIF rV >= (vNoDischarge -0.3) AND rV <(vGaugeOff -0.3)   THEN
	IG.eState := Starting;
	IG.rPRESS := LREAL_TO_REAL(EXPT(10,((rV-vBase)/vSlope+LOG(pBase))));
ELSIF rV >= (vGaugeOff -0.3) THEN
	IG.eState := Off;
	IG.rPRESS := LREAL_TO_REAL(EXPT(10,((rV-vBase)/vSlope+LOG(pBase))));
ELSE
	IG.eState := OoR;
	IG.rPRESS := LREAL_TO_REAL(EXPT(10,((rV-vBase)/vSlope+LOG(pBase))));
END_IF


(* Ion Gauge Protection Functions *)
(* If the PG pressure is greater than the VG.PRO_SP then the gauge is disabled *)
(* If the PG pressure is less than the VG.PRO_SP then the gauge is enabled *)
(* This FB also implements some hysteresis so the gauge doesn't have rapid power cycling while near the turn on boundary *)


IF PG.rPRESS <= IG.rPRO_SP AND PG.xPRESS_OK THEN

	IG.q_xHV_DIS := IG.xHV_SW;
	IG.xILKOk := TRUE;
ELSIF IG.q_xHV_DIS THEN
	IF IG.rPRESS > (IG.rPRO_SP + IG.rHYS_PR)  OR PG.rPRESS > (IG.rPRO_SP + IG.rHYS_PR) THEN
		IG.q_xHV_DIS := FALSE;
		IG.xHV_SW := FALSE;
	END_IF
ELSE
	IG.q_xHV_DIS := FALSE;
	IG.xHV_SW := FALSE;
	IG.xILKOk := FALSE;
END_IF

(* Pressure gauge OK checks *)

GaugeTurnOnTmr(IN:=IG.q_xHV_DIS, PT:=T#10S, Q=>IG.xTurnOnTime);


//Backwards compatibility
IG.xPRESS_OK := (IG.eState = Valid) OR IG.xBAKEOUT;

(* Setpoint evaluation *)
IG.xAT_VAC := (IG.xPRESS_OK AND (IG.rPRESS < IG.rVAC_SP)) OR IG.xBAKEOUT AND (IG.eState = Valid) ;

ACT_Logger();
(*Soft IO Linking*)
// check ethercat Diagnostics
IO();

ACTION ACT_Logger:
IF (IG.xLog) THEN
// ILK logger
IF NOT IG.xILKOk AND NOT IG.q_xHV_DIS THEN
 		fbLogger(sMsg:='Lost external interlock while gauge was on.', eSevr:=TcEventSeverity.Critical);  	
END_IF


// Log Action
tAction(CLK:=  IG.q_xHV_DIS);
IF tAction.Q THEN fbLogger(sMsg:='Ion gauge commanded to switch on', eSevr:=TcEventSeverity.Info); END_IF



//STATE Logger  
IF ePrevState <> IG.eState THEN
	  CASE IG.eState OF
		ValidHi:
			fbLogger(sMsg:='Gauge pressure valid high.', eSevr:=TcEventSeverity.Info);
		ValidLo:
			fbLogger(sMsg:='Gauge pressure valid low.', eSevr:=TcEventSeverity.Info);
		Valid:
			fbLogger(sMsg:='Gauge pressure valid.', eSevr:=TcEventSeverity.Info);
  		GaugeDisconnected:
			fbLogger(sMsg:='Gauge Disconnected.', eSevr:=TcEventSeverity.Critical);
		PressInvalid:
			fbLogger(sMsg:='Gauge pressure invalid.', eSevr:=TcEventSeverity.Warning);
		OoR:
			fbLogger(sMsg:='Gauge pressure out of range.', eSevr:=TcEventSeverity.Warning);
		Starting:
			fbLogger(sMsg:='Gauge starting.', eSevr:=TcEventSeverity.Info);
	  END_CASE
	  ePrevState := IG.eState;  
  END_IF
END_IF
END_ACTION

ACTION IO:
(*soft link inputs*)
IG.i_iPRESS_R:=	i_iPRESS_R; 
(*soft link outputs*)
q_xHV_DIS := IG.q_xHV_DIS;

IG.sPath := sPath;
END_ACTION

METHOD M_HVE : BOOL
VAR_INPUT
		enable:bool; // set to true to enable, false to disable;
END_VAR

this^.IG.xHV_SW:= NOT(enable);
END_METHOD

END_FUNCTION_BLOCK

// POUs/Functions/Deprecated/Valves/FB_VCC_NO
(*Deprecated*)
(* This Function Block Implements Basic Functionality for NO Vent Valves VVC *)
(* Note Interlock Logic is External *)
{attribute 'obsolete' := 'FB_VCC_NO has been deprecated and is not valid!'}
FUNCTION_BLOCK FB_VCC_NO
VAR_IN_OUT
	{attribute 'pytmc' := 'pv:'}
	iq_stValve : ST_VCC_NO;

END_VAR
VAR_INPUT
	i_xExtILK_OK:BOOL; (*Other External Interlock, Set to True when no external interlock is required*)
	i_xOverrideMode : BOOL; (*To be linked to global override bit. This Overrides Vacuum logic only, EPS, MPS and PMPS are still enforces*)

END_VAR
VAR_OUTPUT
END_VAR
VAR

	tonOvrd	:	TON;
	tonDelOK : TON;
	rtOK	:	R_TRIG;
	(*IO*)
	xCLS_DO	AT%Q*: BOOL;

END_VAR


IF NOT iq_stValve.xCLS_OK THEN
iq_stValve.pv_xCLS_SW := FALSE;
END_IF

(* Override logic *)
(* Goal: give ability to override, but do so in a way that people won't forget it.
Solution: Override only after ten seconds of override, protect against blips,
when the valve permission goes true for more than ten seconds consistently, remove override
*)

tonDelOK(IN:=iq_stValve.xCLS_OK, PT:=T#10S);
rtOK(CLK:=tonDelOK.Q);
IF rtOK.Q THEN iq_stValve.pv_xOvrdCls :=FALSE; END_IF

//Override timer
tonOvrd(IN:=iq_stValve.pv_xOvrdCls, PT:=T#10S);

(* Here's where the valve is closed *)
iq_stValve.xCLS_DO := (iq_stValve.pv_xCLS_SW AND iq_stValve.xCLS_OK) OR (tonOvrd.Q AND i_xOverrideMode);

ACTION ACT_IO:
(*inputs*)
iq_stValve.xOverrideMode := i_xOverrideMode;
(*outputs*)
xCLS_DO:= iq_stValve.xCLS_DO;
END_ACTION

METHOD M_Close : BOOL
VAR_INPUT
		close:BOOL; //True to CLose, False to OPEN
END_VAR
This^.iq_stValve.pv_xCLS_SW :=Close;
END_METHOD

END_FUNCTION_BLOCK

// POUs/Functions/Deprecated/Gauges/FB_PressureState
(*Deprecated*)
FUNCTION_BLOCK FB_PressureState
VAR_INPUT
	i_rV	:	REAL;
	i_rVMin	:	REAL := 0.01; // Anything less than this voltage is considered disconnected
	i_rVMax :	REAL := 10.5; // Anything more than this is considered invalid
	i_IGTurnOnTime	:	TIME := T#10S;
	
	i_MinPressure	:	REAL;
	i_MaxPressure	:	REAL;
END_VAR
VAR_OUTPUT
	q_eState 	:	E_PressureState;
END_VAR
VAR_IN_OUT
	iq_stVG	:	ST_VG;
END_VAR
VAR
	tonGaugeTurnOnTmr : TON;
END_VAR

(* Pressure State Evaluation
A. Wallace, 2016-8-31

This FB serves to evaluate the state of the pressure based on the raw voltage, pressure, and gauge state.

*)
// Is the gauge plugged in, and within a reasonable range?
IF i_rV < i_rVMin THEN
	q_eState := GaugeDisconnected;
ELSIF i_rV > i_rVMax THEN
	q_eState := PressInvalid;
ELSE
	// Is the gauge reading back a pressure that makes sense?
	CASE iq_stVG.eTYPE OF
		IG903:
			tonGaugeTurnOnTmr(IN:=iq_stVG.q_xHV_DIS, PT:=i_IGTurnOnTime, Q=>iq_stVG.xTurnOnTime);
			IF iq_stVG.q_xHV_DIS THEN
				IF tonGaugeTurnOnTmr.Q THEN
					IF iq_stVG.rPRESS >= i_MinPressure AND iq_stVG.rPRESS <= i_MaxPressure THEN
						q_eState := Valid;
					ELSE
						q_eState := OoR; 
					END_IF
				ELSE
						q_eState := Starting;
				END_IF
			ELSE
				q_eState := Off;
			END_IF
		IG909:
			IF iq_stVG.q_xHV_DIS THEN
				IF iq_stVG.rPRESS >= i_MinPressure AND iq_stVG.rPRESS <= i_MaxPressure THEN
					q_eState := Valid;
				ELSE
					q_eState := OoR;
				END_IF
			ELSE
				q_eState := Off;
			END_IF
		PG907, PG925, PG722B:
			IF iq_stVG.rPRESS >= i_MinPressure AND iq_stVG.rPRESS <= i_MaxPressure THEN
				q_eState := Valid;
			ELSIF iq_stVG.rPRESS < i_MinPressure THEN
				q_eState := ValidLo;
			ELSE
				q_eState := ValidHi;
			END_IF
		ELSE
			q_eState := PressInvalid;
	END_CASE
END_IF


iq_stVG.eState := q_eState;

// Legacy Press OK boolean eval
iq_stVG.xPRESS_OK := q_eState >= gc_GaugeValidState;

END_FUNCTION_BLOCK

// POUs/Functions/Deprecated/Valves/FB_VCC
(*Deprecated*)
(* THE FB_VCC FUNCTION BLOCK IS DEPRECATED. USE FB_VVC INSTEAD. *)
(* This Function Block Implements Basic Functionality for Vent Valves VVC *)
(* Note Interlock Logic is External *)
FUNCTION_BLOCK FB_VCC
VAR_IN_OUT

END_VAR
VAR_INPUT
	i_xExtILK_OK:BOOL; (*Other External Interlock, Set to True when no external interlock is required*)
	i_xOverrideMode : BOOL; (*To be linked to global override bit. This Overrides Vacuum logic only*)
END_VAR
VAR_OUTPUT
	{attribute 'pytmc' := '
    pv:
	'}
	iq_stValve : ST_VVC;
END_VAR
VAR

	tonOvrd	:	TON;
	tonDelOK : TON;
	rtOK	:	R_TRIG;

	(*IO*)
	q_xOPN_DO	AT%Q*: BOOL;

END_VAR


iq_stValve.xOPN_OK := i_xExtILK_OK;

IF NOT iq_stValve.xOPN_OK THEN
iq_stValve.pv_xOPN_SW := FALSE;
END_IF

(* Override logic *)
(* Goal: give ability to override, but do so in a way that people won't forget it.
Solution: Override only after ten seconds of override, protect against blips,
when the valve permission goes true for more than ten seconds consistently, remove override
*)

tonDelOK(IN:=iq_stValve.xOPN_OK, PT:=T#10S);
rtOK(CLK:=tonDelOK.Q);
IF rtOK.Q THEN iq_stValve.xOvrdOpn :=FALSE; END_IF

//Override timer
tonOvrd(IN:=iq_stValve.xOvrdOpn, PT:=T#10S);

(* Here's where the valve opens *)
iq_stValve.q_xOPN_DO := (iq_stValve.pv_xOPN_SW AND iq_stValve.xOPN_OK) OR (tonOvrd.Q AND i_xOverrideMode);

(*IO Mapping*)
ACT_IO();

ACTION ACT_IO:
(*inputs*)
iq_stValve.xOverrideMode := i_xOverrideMode;
(*outputs*)
q_xOPN_DO:= iq_stValve.q_xOPN_DO;
END_ACTION

METHOD PUBLIC M_IsClosed : BOOL
VAR_INPUT
END_VAR
M_IsClosed := NOT This^.q_xOPN_DO;
END_METHOD

METHOD PUBLIC M_IsOpen : BOOL
VAR_INPUT
END_VAR
M_IsOpen := This^.q_xOPN_DO;
END_METHOD

// Use this Methode to Open or close the valve by setting the OPN_SW to the input value.
METHOD PUBLIC M_Set_OPN_SW : BOOL
VAR_INPUT
		value:BOOL;  //True to SET, False to RESET
END_VAR
This^.iq_stValve.pv_xOPN_SW := value;
END_METHOD

END_FUNCTION_BLOCK

// POUs/Functions/Valves/FB_VVC
(* This Function Block Implements Basic Functionality for Vent Valves VVC.

	This function block is also intended for the general use case of solenoid driven (non-variable) valves that lack status readbacks or position indicators. 
*)
(* Note Interlock Logic is External *)
FUNCTION_BLOCK FB_VVC
VAR_IN_OUT

END_VAR
VAR_INPUT
	i_xExtILK_OK:BOOL; (*Other External Interlock, Set to True when no external interlock is required*)
	i_xOverrideMode : BOOL; (*To be linked to global override bit. This Overrides Vacuum logic only*)
END_VAR
VAR_OUTPUT
	{attribute 'pytmc' := '
    pv:
	'}
	iq_stValve : ST_VVC;
END_VAR
VAR

	tonOvrd	:	TON;
	tonDelOK : TON;
	rtOK	:	R_TRIG;

	(*IO*)
	q_xOPN_DO	AT%Q*: BOOL;

	pv_xOvrdOpn: INT;
END_VAR


iq_stValve.xOPN_OK := i_xExtILK_OK;

IF NOT iq_stValve.xOPN_OK THEN
iq_stValve.pv_xOPN_SW := FALSE;
END_IF

(* Override logic *)
(* Goal: give ability to override, but do so in a way that people won't forget it.
Solution: Override only after ten seconds of override, protect against blips,
when the valve permission goes true for more than ten seconds consistently, remove override
*)

tonDelOK(IN:=iq_stValve.xOPN_OK, PT:=T#10S);
rtOK(CLK:=tonDelOK.Q);
IF rtOK.Q THEN iq_stValve.xOvrdOpn :=FALSE; END_IF
// Release the Force Open bit when the system override is false
IF NOT (i_xOverrideMode) THEN  iq_stValve.xOvrdOpn :=FALSE; END_IF

//Override timer
tonOvrd(IN:=iq_stValve.xOvrdOpn, PT:=T#10S);

(* Here's where the valve opens *)
iq_stValve.q_xOPN_DO := (iq_stValve.pv_xOPN_SW AND iq_stValve.xOPN_OK) OR (tonOvrd.Q AND i_xOverrideMode);

(*IO Mapping*)
ACT_IO();

ACTION ACT_IO:
(*inputs*)
iq_stValve.xOverrideMode := i_xOverrideMode;
(*outputs*)
q_xOPN_DO:= iq_stValve.q_xOPN_DO;
END_ACTION

// Method Returns True if the Valve is closed, i.e. the open digital output is not active
METHOD PUBLIC M_IsClosed : BOOL
VAR_INPUT
END_VAR
M_IsClosed := NOT This^.q_xOPN_DO;
END_METHOD

// Method Returns True if the Valve is open, i.e. the open digital output is active
METHOD PUBLIC M_IsOpen : BOOL
VAR_INPUT
END_VAR
M_IsOpen := This^.q_xOPN_DO;
END_METHOD

METHOD PUBLIC M_Open : BOOL
VAR_INPUT
	open: bool; //Set to true to open the valvue, false to close
END_VAR
This^.iq_stValve.pv_xOPN_SW := open;
END_METHOD

// Use this Methode to Open or close the valve by setting the OPN_SW to the input value.
METHOD PUBLIC M_Set_OPN_SW : BOOL
VAR_INPUT
	value:BOOL; //True to SET, False to RESET
END_VAR
This^.iq_stValve.pv_xOPN_SW := value;
END_METHOD

END_FUNCTION_BLOCK

// POUs/Functions/Deprecated/Valves/FB_VGC_AP
(*Deprectated*)
(* This function block implements basic functionality for Isolation Gate Valves with Appertures*)
(* This function block interlock is as follows:
1. The valve can be opened when the difference between the pressures on both sides is
less than the maximum differential pressure.
2. This rule persists until the pressures on both sides are lower than the vacuum-setpoint.
3. Once at-vac, the valve will close if the pressure on either side rises above the setpoint.*)
(*This function block also implements PMPS and EPS interlocks, as well as Fast MPS trigger*)
(* MPS is triggered differently than the VGC *)
{attribute 'no_check'}
{attribute 'obsolete' := 'FB_VGC_AP has been deprecated and is not valid!'}
FUNCTION_BLOCK FB_VGC_AP
VAR_IN_OUT
	
END_VAR
VAR_INPUT
	(*Upstream Gauge, usually ion gauge*)
	i_stUSG	:	ST_VG;
	(*Downstream Gauge, usually ion gauge*)
	i_stDSG	:	ST_VG;
	{attribute 'pytmc' := '
    pv: Dis_DPIlk
	'}
	i_xDis_DPIlk : BOOL := FALSE;  (* Set to true when calling the function to disable the differential pressure interlock *)
	{attribute 'pytmc' := '
    pv: EPS_OK
	'}
	i_xEPS_OK:	BOOL	:= TRUE; (*External EPS interlock, Set to TRUE when no EPS interlock is required, otherwise set to correct interlock signal*)
	{attribute 'pytmc' := '
    pv: MPS_OK
	'}
	i_xPMPS_OK:	BOOL	; (*External MPS interlock, Set to TRUE when no PMPS interlock is required*)
	i_xExt_OK: BOOL; (*Other External Interlock, Set to True when no external interlock is required. If this Valve is neigboring a Fast Shutter this should be linked to the fast shutter xVAC_FAULT_OK*)
	i_xOverrideMode : BOOL; (*To be linked to global override bit. This Overrides Vacuum logic only, EPS, MPS and PMPS are still enforces*)
	// Reset fault
	{attribute 'pytmc' := '
    pv: FF_Reset
	'}
    i_xReset: BOOL;
	i_sDevName : T_MaxString :=  'VGC'; // Device name for diagnostic
END_VAR
VAR_OUTPUT
	{attribute 'pytmc' := '
    pv:
	'}
	iq_stValve : ST_VGC; (* All valve data and states will be in this struct*)
	
	{attribute 'pytmc' := '
    pv: MPS_FAULT_OK
	'}
	xMPS_OK:	BOOL; (*MPS Fast OK, is set when the Valve is Open*)
END_VAR
VAR_IN_OUT
	io_fbFFHWO    :    FB_HardwareFFOutput;
END_VAR
VAR
	// PMPS
	fbFF    :    FB_FastFault :=(
        i_DevName := 'VGC Aptr',
        i_Desc := 'Fault occurs when the valve is not in open state',
        i_TypeCode := 16#1010);
	//g_FastFaultOutput1	:	FB_HardwareFFOutput;	

	{attribute 'instance-path'}
	{attribute 'noinit'}
	sPath: STRING;
	
	rDiffPressAllowed	:	REAL := 22.5; // Torr, Default value comes from Vat Valve Manual
	rDiffPress : REAL;
	set : BOOL;
    reset: BOOL;
	  
	xFirstPass	:	BOOL;
	fbFSInit		:	R_TRIG;
	
	tonDelOK : TON;
	rtOK	:	R_TRIG;
	tonOvrd	:	TON;
	
	tDelOK	:	TIME := T#60S;
	tOvrd	:	TIME := T#10s;
	
	
	(* Timeouts*)
	tTimeOutDuration: TIME:= T#30S;
	tOPNtimeout: TON;
	tCLStimeout:TON;
	
	 // For logging
    fbLogger : FB_LogMessage := (eSubsystem:=E_SubSystem.VACUUM);
    ePrevState : E_VGC;
    tErrorPresent : R_TRIG;
    tAction : R_TRIG; // Primary action of this device (OPN_DO, PUMP_RUN, etc.)
    tOverrideActivated : R_TRIG;
	
	
	
	(*IO*)
	i_xOpnLS	AT%I*: BOOL;
	i_xClsLS	AT%I*: BOOL;
	q_xOPN_DO	AT%Q*: BOOL;
	
END_VAR

(* Vacuum gate valve
A. Wallace
16-10-29

A gate valve isolates vacuum volumes. Ideally it can be opened when a system is vented
to allow for faster pumping, and will close when high vacuum is lost.

The following behavior is good for valves in something like a gas attenuator.
This function block does the following:
1. The valve can be opened when the difference between the pressures on both sides is
less than the maximum differential pressure.
2. This rule persists until the pressures on both sides are lower than the vacuum-setpoint.
3. Once at-vac, the valve will close if the pressure on either side rises above the setpoint.

Alternatively, the differential pressure interlock can be disabled so the valve may only be opened
if the pressure on both sides is lower than the at-vacuum-setpoint. You want this behavior if 
the valve is to be used in a UHV section.

Hysteresis is employed to ensure a smooth transition from vented/pumping down, to at-vac.

Finally, an override system is built in so you can bypass all the interlocking logic and 
get back online.
*)
(* 10/1/2018 Margaret Ghaly included EPS, PMPS Checkes and MPS trigger signals*)


fbFSInit( CLK := TRUE, Q => xFirstPass);
(*IO Mapping*)
ACT_IO();

(* On first PLC pass, put valve into vented state, which implies a closed valve *)
IF xFirstPass THEN
	iq_stValve.eVGC_State := Vented;
	iq_stValve.pv_xOPN_SW := FALSE;
	fbFF.i_DevName := i_sDevName;
END_IF


///Check valve position
IF iq_stValve.i_xClsLS AND  iq_stValve.i_xOpnLS THEN
	iq_stValve.eState:=INVALID;
ELSIF NOT iq_stValve.i_xClsLS AND iq_stValve.i_xOpnLS AND iq_stValve.q_xOPN_DO THEN 
	iq_stValve.eState:=OPEN;
ELSIF NOT iq_stValve.i_xClsLS AND iq_stValve.i_xOpnLS AND NOT iq_stValve.q_xOPN_DO THEN 
	iq_stValve.eState:=OPEN_F;
ELSIF iq_stValve.i_xClsLS AND NOT iq_stValve.i_xOpnLS AND NOT iq_stValve.q_xOPN_DO THEN 
	iq_stValve.eState:=CLOSED;
ELSIF NOT iq_stValve.i_xClsLS AND NOT iq_stValve.i_xOpnLS THEN 
	iq_stValve.eState:=MOVING;
ELSE
	iq_stValve.eState:=INVALID;
END_IF

// Update hysteresis
///////////////////////////////////////////////////
IF iq_stValve.rAT_VAC_SP_LAST <> iq_stValve.rAT_VAC_SP OR xFirstPass THEN
	iq_stValve.rAT_VAC_SP_LAST := iq_stValve.rAT_VAC_SP;
	iq_stValve.rAT_VAC_HYS := iq_stValve.rHYST_PERC * iq_stValve.rAT_VAC_SP;
END_IF

iq_stValve.rAT_VAC_HYS := LIMIT(0, iq_stValve.rAT_VAC_HYS, iq_stValve.rAT_VAC_SP);
IF iq_stValve.rAT_VAC_SP <> 0 THEN
	IF iq_stValve.rHYST_PERC <> (iq_stValve.rAT_VAC_HYS / iq_stValve.rAT_VAC_SP) THEN
		iq_stValve.rHYST_PERC := LIMIT(0, (iq_stValve.rAT_VAC_HYS / iq_stValve.rAT_VAC_SP) ,1);
	END_IF

END_IF
// Valve at vacuum check
///////////////////////////////////////////////////
	set := i_stUSG.rPRESS < iq_stValve.rAT_VAC_HYS AND i_stDSG.rPRESS < iq_stValve.rAT_VAC_HYS AND i_stUSG.xPRESS_OK AND i_stDSG.xPRESS_OK;
 	iq_stValve.xAT_VAC S= set;
	reset := i_stUSG.rPRESS > iq_stValve.rAT_VAC_SP OR i_stDSG.rPRESS > iq_stValve.rAT_VAC_SP OR NOT i_stUSG.xPRESS_OK OR NOT i_stDSG.xPRESS_OK;
	iq_stValve.xAT_VAC R= reset;
	
// Differential pressure check
///////////////////////////////////////////////////
	(* Calc the differential pressure across the valve *)
	rDiffPress := ABS(i_stUSG.rPRESS - i_stDSG.rPRESS);
	
	(* As long as the differential pressure is less than 30mbar, the valve is allowed to open *)
	IF rDiffPress <= rDiffPressAllowed AND i_stUSG.xPRESS_OK AND i_stDSG.xPRESS_OK THEN
		iq_stValve.xDP_OK := TRUE;
	ELSE
		iq_stValve.xDP_OK	:= FALSE;
		(* If the differential pressure is exceeded, even when the valve is open,
		the state is unexpected and triggers a fault, because it suggests that something
		is wrong with the valve, or gauges or mapping or there is a major leak on one side.*)
		iq_stValve.eVGC_State := ERR_DiffPress;
	END_IF

// Valve state
///////////////////////////////////////////////////
CASE iq_stValve.eVGC_State OF
	Vented: (* The Vented state is used during pump down *)
        //Log new state
        IF ePrevState <> iq_stValve.eVGC_State THEN
            fbLogger(sMsg:='Vented', eSevr:=TcEventSeverity.Info);
            ePrevState := iq_stValve.eVGC_State;
		END_IF
        
		(* Assuming the pump down went well, we are now at vacuum on both sides,
		so we move to the vacuum state, otherwise remain in the vented state *)
		IF iq_stValve.xAT_VAC AND (NOT (iq_stValve.xERR_DifPres)) AND  (NOT (iq_stValve.xERR_SP)) and  (NOT (iq_stValve.xERR_ExtFault))THEN
		    iq_stValve.eVGC_State := AtVacuum;
		ELSE
		    iq_stValve.eVGC_State := Vented;
		END_IF
	
	AtVacuum:
        //Log new state
        IF ePrevState <> iq_stValve.eVGC_State THEN
            fbLogger(sMsg:='Vacuum setpoint satisfied', eSevr:=TcEventSeverity.Info);
            ePrevState := iq_stValve.eVGC_State;
		END_IF
        
		IF iq_stValve.xAT_VAC THEN
		(* If both pressure setpoints are made,
		then enable the differential pressure interlock, regardless of the valve state
		assuming we're using some kind of ion gauge where a pressure setpoint cannot be higher than 1E-4 T *)
		iq_stValve.eVGC_State := AtVacuum;
				
		ELSE
		
			(* If the valve is open (or in an unknown state) and either gauge is not at it's vacuum setpoint,
			we have a loss of vacuum error *)
			IF (iq_stValve.i_xOpnLS OR (NOT iq_stValve.i_xOpnLS AND NOT iq_stValve.i_xClsLS)) THEN
				iq_stValve.eVGC_State := ERR_LostVac;
				iq_stValve.xERR_SP := TRUE; //TAW changed this to the ERR_SP bool because I think that's what it was intended to be?
		
			(* Alternatively, if the valve is already closed and we lose pressure on one side,
			it was probably intentional venting, so we calmly move back to venting mode, and
			disable the differential pressure interlock *) //?? 
			ELSIF iq_stValve.i_xClsLS THEN
				iq_stValve.eVGC_State := Vented;
			END_IF
		
		END_IF
	ERR_DiffPress:
        //Log new state
        IF ePrevState <> iq_stValve.eVGC_State THEN
            fbLogger(sMsg:='Potential accidental vent.', eSevr:=TcEventSeverity.Critical);
            ePrevState := iq_stValve.eVGC_State;
		END_IF
        
		IF NOT (iq_stValve.xERR_DifPres) THEN
			iq_stValve.eVGC_State := Vented;
		END_IF
		
	
	ERR_LostVac:
        //Log new state
        IF ePrevState <> iq_stValve.eVGC_State THEN
            fbLogger(sMsg:='Unexpected loss of vacuum while valve was open.', eSevr:=TcEventSeverity.Critical);
            ePrevState := iq_stValve.eVGC_State;
		END_IF
		IF NOT (iq_stValve.xERR_SP) THEN
			iq_stValve.eVGC_State := Vented;
		END_IF
		
	ERR_ExtFault:
        //Log new state
        IF ePrevState <> iq_stValve.eVGC_State THEN
            fbLogger(sMsg:='Lost external interlock while valve was open.', eSevr:=TcEventSeverity.Critical);
            ePrevState := iq_stValve.eVGC_State;
		END_IF
		IF NOT (iq_stValve.xERR_ExtFault) AND (NOT i_xExt_OK) THEN
			iq_stValve.eVGC_State := Vented;
		END_IF
	END_CASE



IF (NOT i_xExt_OK) THEN
	iq_stValve.eVGC_State := ERR_ExtFault;
	iq_stValve.xERR_ExtFault := TRUE;
END_IF

// Interlock evaluation - with bypass for DP ILK bypass
///////////////////////////////////////////////
IF i_xDis_DPIlk THEN
	iq_stValve.xOPN_OK := iq_stValve.xEXT_OK; // AND iq_stValve.xDP_OK ;
ELSE
	iq_stValve.xOPN_OK := iq_stValve.xEXT_OK AND iq_stValve.xAT_VAC;
END_IF


(* Valve operation *)

(* Override logic *)
(* Goal: give ability to override, but do so in a way that people won't forget it.
Solution: Override only after ten seconds of override, protect against blips,
when the valve permission goes true for more than ten seconds consistently, remove override
*)

tonDelOK(IN:=iq_stValve.xOPN_OK, PT:=tDelOK);
rtOK(CLK:=tonDelOK.Q);
IF rtOK.Q AND iq_stValve.pv_xOvrdOpn THEN 
	iq_stValve.pv_xOvrdOpn :=FALSE;
	if (iq_stValve.eState = OPEN) AND (i_xOverrideMode) THEN iq_stValve.pv_xOPN_SW := TRUE; END_IF  //for seamless transition
	//Log
    fbLogger(sMsg:='Override expired', eSevr:=TcEventSeverity.Warning);
    
END_IF

//Override timer
tonOvrd(IN:=iq_stValve.pv_xOvrdOpn, PT:=tOvrd);

(* If Epics Command to close the Valve, check if PMPS and EPS are ok, otherwise Keep command set to open valve *)
IF NOT(iq_stValve.pv_xOPN_SW) AND ((NOT i_xPMPS_OK) OR (NOT i_xEPS_OK)) THEN
	//iq_stValve.pv_xOPN_SW := TRUE; // plc to only reset never to set this signal
END_IF
(* Reset the EPICS command to open the valve if the interlock is lost *) 
(* based on EPS ok state, EPS overrides OPN_OK*)
IF NOT iq_stValve.xOPN_OK THEN
	IF i_xEPS_OK THEN iq_stValve.pv_xOPN_SW := FALSE; iq_stValve.sErrorMessage := 'ILK Active';
	ELSE //iq_stValve.pv_xOPN_SW := TRUE;		// plc to only reset never to set this signal
	END_IF
END_IF

(* Here's where the valve opens *)
iq_stValve.q_xOPN_DO := (iq_stValve.pv_xOPN_SW AND iq_stValve.xOPN_OK) OR (tonOvrd.Q AND i_xOverrideMode);

(* When the valve  is open MPS is OK*)
xMPS_OK := i_xOpnLS XOR i_xClsLS;

///Check valve moving postion timout
IF NOT iq_stValve.i_xClsLS AND tCLStimeout.Q THEN 
	iq_stValve.bErrorPresent := TRUE;
	iq_stValve.sErrorMessage := 'Close Timeout';
ELSIF NOT iq_stValve.i_xOpnLS AND tOPNtimeout.Q THEN 
	iq_stValve.bErrorPresent := TRUE; 
	iq_stValve.sErrorMessage := 'Open Timeout';
END_IF
IF (iq_stValve.eState=INVALID) THEN
	iq_stValve.bErrorPresent := TRUE; 
	iq_stValve.sErrorMessage := CONCAT(sPath,'Invalid Valve Position');
END_IF
(*Timers*)
tOPNtimeout(IN:= iq_stValve.q_xOPN_DO, PT := tTimeOutDuration );
tCLStimeout(IN:= NOT iq_stValve.q_xOPN_DO, PT := tTimeOutDuration);


// Log valve timeouts
tErrorPresent(CLK:=iq_stValve.bErrorPresent);
IF tErrorPresent.Q THEN fbLogger(sMsg:=iq_stValve.sErrorMessage, eSevr:=TcEventSeverity.Warning); END_IF

// Log valve open
tAction(CLK:= iq_stValve.q_xOPN_DO);
IF tAction.Q THEN fbLogger(sMsg:='Valve commanded open', eSevr:=TcEventSeverity.Info); END_IF

// Log override mode enabled
tOverrideActivated(CLK:= (tonOvrd.Q AND i_xOverrideMode));
IF tOverrideActivated.Q THEN fbLogger(sMsg:='Valve override mode activated', eSevr:=TcEventSeverity.Warning); END_IF


// Alarm reset
//////////////////////////////////////
ACT_ResetAlarms();

(*IO Mapping*)
ACT_IO();

(*FAST FAULT*)
fbFF(i_xOK := xMPS_OK,
    i_xReset := i_xReset,
	i_xAutoReset :=TRUE,
    io_fbFFHWO := io_fbFFHWO);

ACTION ACT_IO:
(*inputs*)
iq_stValve.i_xOpnLS := 	i_xOpnLS;
iq_stValve.i_xClsLS:=	i_xClsLS;
iq_stValve.xEXT_OK := i_xEXT_OK;
iq_stValve.xOverrideMode := i_xOverrideMode;
(*outputs*)
q_xOPN_DO:= iq_stValve.q_xOPN_DO;
END_ACTION

ACTION ACT_ResetAlarms:
iq_stValve.xERR_DifPres R= iq_stValve.pv_xAlmRst;
iq_stValve.xERR_SP R= iq_stValve.pv_xAlmRst;
iq_stValve.bErrorPresent R= iq_stValve.pv_xAlmRst;

IF ( iq_stValve.pv_xAlmRst) THEN
	iq_stValve.sErrorMessage :='';
END_IF
END_ACTION

METHOD PUBLIC M_IsClosed : BOOL
VAR_INPUT
END_VAR
M_IsClosed := (This^.iq_stValve.eState = E_ValvePositionState.CLOSED);
END_METHOD

METHOD PUBLIC M_IsOpen : BOOL
VAR_INPUT
END_VAR
M_IsOpen := (This^.iq_stValve.eState = E_ValvePositionState.OPEN);
END_METHOD

// Use this Methode to Open or close the valve by setting the OPN_SW to the input value.
METHOD PUBLIC M_Set_OPN_SW : BOOL
VAR_INPUT
		value:BOOL;
END_VAR
This^.iq_stValve.pv_xOPN_SW := value;
END_METHOD

END_FUNCTION_BLOCK

// POUs/Functions/Deprecated/Valves/FB_VGC_EBD
(*Deprecated*)
(* This function block is similar to the FB_VGC, except it has 2 outputs to actuate the Valve*)
(* This function block implements basic functionality for Isolation Gate Valves*)
(* This function block interlock is as follows:
1. The valve can be opened when the difference between the pressures on both sides is
less than the maximum differential pressure.
2. This rule persists until the pressures on both sides are lower than the vacuum-setpoint.
3. Once at-vac, the valve will close if the pressure on either side rises above the setpoint.*)
(*This function block also implements PMPS and EPS interlocks, as well as Fast MPS trigger*)
{attribute 'no_check'}
{attribute 'obsolete' := 'FB_VGC_EBD has been deprecated and is not valid!'}
FUNCTION_BLOCK FB_VGC_EBD
VAR_IN_OUT
	
END_VAR
VAR_INPUT
	(*Upstream Gauge, usually ion gauge*)
	i_stUSG	:	ST_VG;
	(*Downstream Gauge, usually ion gauge*)
	i_stDSG	:	ST_VG;
	{attribute 'pytmc' := '
    pv: Dis_DPIlk
	'}
	i_xDis_DPIlk : BOOL := FALSE;  (* Set to true when calling the function to disable the differential pressure interlock *)
	{attribute 'pytmc' := '
    pv: EPS_OK
	'}
	i_xEPS_OK:	BOOL	:= TRUE; (*External EPS interlock, Set to TRUE when no EPS interlock is required, otherwise set to correct interlock signal*)
	{attribute 'pytmc' := '
    pv: MPS_OK
	'}
	i_xPMPS_OK:	BOOL	; (*External MPS interlock, Set to TRUE when no PMPS interlock is required*)
	i_xExt_OK: BOOL; (*Other External Interlock, Set to True when no external interlock is required*)
	i_xOverrideMode : BOOL; (*To be linked to global override bit. This Overrides Vacuum logic only, EPS, MPS and PMPS are still enforces*)
	// Reset fault
	{attribute 'pytmc' := '
    pv: FF_Reset
	'}
    i_xReset: BOOL;
	i_sDevName : T_MaxString :=  'VGC'; // Device name for diagnostic
END_VAR
VAR_OUTPUT
	{attribute 'pytmc' := '
    pv:
	'}
	iq_stValve : ST_VGC; (* All valve data and states will be in this struct*)
	
	{attribute 'pytmc' := '
    pv: MPS_FAULT_OK
	field: ZNAM MPS FAULT ;
	field: ONAM MPS OK ;
	'}
	xMPS_OK:	BOOL; (*MPS Fast OK, is set when the Valve is Open*)
END_VAR
VAR_IN_OUT
	io_fbFFHWO    :    FB_HardwareFFOutput;
END_VAR
VAR
	// PMPS
	fbFF    :    FB_FastFault :=(
        i_DevName := 'VGC',
        i_Desc := 'Fault occurs when the valve is not in open state',
        i_TypeCode := 16#1010);
	{attribute 'instance-path'}
	{attribute 'noinit'}
	sPath: STRING;
	
	rDiffPressAllowed	:	REAL := 22.5; // Torr, Default value comes from Vat Valve Manual
	rDiffPress : REAL;
	set : BOOL;
    reset: BOOL;
	  
	xFirstPass	:	BOOL;
	fbFSInit		:	R_TRIG;
	
	tonDelOK : TON;
	rtOK	:	R_TRIG;
	tonOvrd	:	TON;
	
	tDelOK	:	TIME := T#60S;
	tOvrd	:	TIME := T#10s;
	
	
	(* Timeouts*)
	tTimeOutDuration: TIME:= T#30S;
	tOPNtimeout: TON;
	tCLStimeout:TON;
	
	
	 // For logging
    fbLogger : FB_LogMessage := (eSubsystem:=E_SubSystem.VACUUM);
    ePrevState : E_VGC;
    tErrorPresent : R_TRIG;
    tAction : R_TRIG; // Primary action of this device (OPN_DO, PUMP_RUN, etc.)
    tOverrideActivated : R_TRIG;
	
	(*IO*)
	i_xOpnLS	AT%I*: BOOL;
	i_xClsLS	AT%I*: BOOL;
	q_xOPN_DO	AT%Q*: BOOL;
	q_xOPN_DO_2	AT%Q*: BOOL;
	
END_VAR

(* Vacuum gate valve
A. Wallace
16-10-29

A gate valve isolates vacuum volumes. Ideally it can be opened when a system is vented
to allow for faster pumping, and will close when high vacuum is lost.

The following behavior is good for valves in something like a gas attenuator.
This function block does the following:
1. The valve can be opened when the difference between the pressures on both sides is
less than the maximum differential pressure.
2. This rule persists until the pressures on both sides are lower than the vacuum-setpoint.
3. Once at-vac, the valve will close if the pressure on either side rises above the setpoint.

Alternatively, the differential pressure interlock can be disabled so the valve may only be opened
if the pressure on both sides is lower than the at-vacuum-setpoint. You want this behavior if 
the valve is to be used in a UHV section.

Hysteresis is employed to ensure a smooth transition from vented/pumping down, to at-vac.

Finally, an override system is built in so you can bypass all the interlocking logic and 
get back online.
*)
(* 10/1/2018 Margaret Ghaly included EPS, PMPS Checkes and MPS trigger signals*)


fbFSInit( CLK := TRUE, Q => xFirstPass);
(*IO Mapping*)
ACT_IO();

(* On first PLC pass, put valve into vented state, which implies a closed valve *)
IF xFirstPass THEN
	iq_stValve.eVGC_State := Vented;
	iq_stValve.pv_xOPN_SW := FALSE;
	fbFF.i_DevName := i_sDevName;
END_IF


///Check valve postion
IF iq_stValve.i_xClsLS AND  iq_stValve.i_xOpnLS THEN
	iq_stValve.eState:=INVALID;
ELSIF NOT iq_stValve.i_xClsLS AND iq_stValve.i_xOpnLS AND iq_stValve.q_xOPN_DO THEN 
	iq_stValve.eState:=OPEN;
ELSIF iq_stValve.i_xClsLS AND NOT iq_stValve.i_xOpnLS AND NOT iq_stValve.q_xOPN_DO THEN 
	iq_stValve.eState:=CLOSED;
ELSIF NOT iq_stValve.i_xClsLS AND NOT iq_stValve.i_xOpnLS THEN 
	iq_stValve.eState:=MOVING;
ELSE
	iq_stValve.eState:=INVALID;
END_IF

// Update hysteresis
///////////////////////////////////////////////////
IF iq_stValve.rAT_VAC_SP_LAST <> iq_stValve.rAT_VAC_SP OR xFirstPass THEN
	iq_stValve.rAT_VAC_SP_LAST := iq_stValve.rAT_VAC_SP;
	iq_stValve.rAT_VAC_HYS := iq_stValve.rHYST_PERC * iq_stValve.rAT_VAC_SP;
END_IF

iq_stValve.rAT_VAC_HYS := LIMIT(0, iq_stValve.rAT_VAC_HYS, iq_stValve.rAT_VAC_SP);
IF iq_stValve.rAT_VAC_SP <> 0 THEN
	IF iq_stValve.rHYST_PERC <> (iq_stValve.rAT_VAC_HYS / iq_stValve.rAT_VAC_SP) THEN
		iq_stValve.rHYST_PERC := LIMIT(0, (iq_stValve.rAT_VAC_HYS / iq_stValve.rAT_VAC_SP) ,1);
	END_IF
	
END_IF
// Valve at vacuum check
///////////////////////////////////////////////////
	set := i_stUSG.rPRESS < iq_stValve.rAT_VAC_HYS AND i_stDSG.rPRESS < iq_stValve.rAT_VAC_HYS AND i_stUSG.xPRESS_OK AND i_stDSG.xPRESS_OK;
 	iq_stValve.xAT_VAC S= set;
	reset := i_stUSG.rPRESS > iq_stValve.rAT_VAC_SP OR i_stDSG.rPRESS > iq_stValve.rAT_VAC_SP OR NOT i_stUSG.xPRESS_OK OR NOT i_stDSG.xPRESS_OK;
	iq_stValve.xAT_VAC R= reset;
	
// Differential pressure check
///////////////////////////////////////////////////
	(* Calc the differential pressure across the valve *)
	rDiffPress := ABS(i_stUSG.rPRESS - i_stDSG.rPRESS);
	
	(* As long as the differential pressure is less than 30mbar, the valve is allowed to open *)
	IF rDiffPress <= rDiffPressAllowed AND i_stUSG.xPRESS_OK AND i_stDSG.xPRESS_OK THEN
		iq_stValve.xDP_OK := TRUE;
	ELSE
		iq_stValve.xDP_OK	:= FALSE;
		(* If the differential pressure is exceeded, even when the valve is open,
		the state is unexpected and triggers a fault, because it suggests that something
		is wrong with the valve, or gauges or mapping or there is a major leak on one side.*)
		iq_stValve.eVGC_State := ERR_DiffPress;
        iq_stValve.xERR_DifPres := TRUE;
	END_IF

// Valve state
///////////////////////////////////////////////////
CASE iq_stValve.eVGC_State OF
	Vented: (* The Vented state is used during pump down *)
        //Log new state
        IF ePrevState <> iq_stValve.eVGC_State THEN
            fbLogger(sMsg:='Vented', eSevr:=TcEventSeverity.Info);
            ePrevState := iq_stValve.eVGC_State;
		END_IF
        
		(* Assuming the pump down went well, we are now at vacuum on both sides,
		so we move to the vacuum state, otherwise remain in the vented state *)
		IF iq_stValve.xAT_VAC AND (NOT (iq_stValve.xERR_DifPres)) AND  (NOT (iq_stValve.xERR_SP)) and  (NOT (iq_stValve.xERR_ExtFault))THEN
		    iq_stValve.eVGC_State := AtVacuum;
		ELSE
		    iq_stValve.eVGC_State := Vented;
		END_IF
	
	AtVacuum:
        //Log new state
        IF ePrevState <> iq_stValve.eVGC_State THEN
            fbLogger(sMsg:='Vacuum setpoint satisfied', eSevr:=TcEventSeverity.Info);
            ePrevState := iq_stValve.eVGC_State;
		END_IF
        
		IF iq_stValve.xAT_VAC THEN
		(* If both pressure setpoints are made,
		then enable the differential pressure interlock, regardless of the valve state
		assuming we're using some kind of ion gauge where a pressure setpoint cannot be higher than 1E-4 T *)
		iq_stValve.eVGC_State := AtVacuum;
				
		ELSE
		
			(* If the valve is open (or in an unknown state) and either gauge is not at it's vacuum setpoint,
			we have a loss of vacuum error *)
			IF (iq_stValve.i_xOpnLS OR (NOT iq_stValve.i_xOpnLS AND NOT iq_stValve.i_xClsLS)) THEN
				iq_stValve.eVGC_State := ERR_LostVac;
				iq_stValve.xERR_SP := TRUE; //TAW changed this to the ERR_SP bool because I think that's what it was intended to be?
		
			(* Alternatively, if the valve is already closed and we lose pressure on one side,
			it was probably intentional venting, so we calmly move back to venting mode, and
			disable the differential pressure interlock *) //?? 
			ELSIF iq_stValve.i_xClsLS THEN
				iq_stValve.eVGC_State := Vented;
			END_IF
		
		END_IF
	
	ERR_DiffPress:
        //Log new state
        IF ePrevState <> iq_stValve.eVGC_State THEN
            fbLogger(sMsg:='Potential accidental vent.', eSevr:=TcEventSeverity.Critical);
            ePrevState := iq_stValve.eVGC_State;
		END_IF
        
		IF NOT (iq_stValve.xERR_DifPres) THEN
			iq_stValve.eVGC_State := Vented;
		END_IF
		
	
	ERR_LostVac:
        //Log new state
        IF ePrevState <> iq_stValve.eVGC_State THEN
            fbLogger(sMsg:='Unexpected loss of vacuum while valve was open.', eSevr:=TcEventSeverity.Critical);
            ePrevState := iq_stValve.eVGC_State;
		END_IF
		IF NOT (iq_stValve.xERR_SP) THEN
			iq_stValve.eVGC_State := Vented;
		END_IF
		
	ERR_ExtFault:
        //Log new state
        IF ePrevState <> iq_stValve.eVGC_State THEN
            fbLogger(sMsg:='Lost external interlock while valve was open.', eSevr:=TcEventSeverity.Critical);
            ePrevState := iq_stValve.eVGC_State;
		END_IF
		IF NOT (iq_stValve.xERR_ExtFault) AND (NOT i_xExt_OK) THEN
			iq_stValve.eVGC_State := Vented;
		END_IF
END_CASE

IF (NOT i_xExt_OK) THEN
	iq_stValve.eVGC_State := ERR_ExtFault;
	iq_stValve.xERR_ExtFault := TRUE;
END_IF

// Interlock evaluation - with bypass for DP ILK bypass
///////////////////////////////////////////////
IF i_xDis_DPIlk THEN
	iq_stValve.xOPN_OK := iq_stValve.xEXT_OK; // AND iq_stValve.xDP_OK ;
ELSE
	iq_stValve.xOPN_OK := iq_stValve.xEXT_OK AND iq_stValve.xAT_VAC;
END_IF


(* Valve operation *)

(* Override logic *)
(* Goal: give ability to override, but do so in a way that people won't forget it.
Solution: Override only after ten seconds of override, protect against blips,
when the valve permission goes true for more than ten seconds consistently, remove override
*)

tonDelOK(IN:=iq_stValve.xOPN_OK, PT:=tDelOK);
rtOK(CLK:=tonDelOK.Q);
IF rtOK.Q AND iq_stValve.pv_xOvrdOpn THEN 
	iq_stValve.pv_xOvrdOpn :=FALSE;
	if (iq_stValve.eState = OPEN) AND (i_xOverrideMode) THEN iq_stValve.pv_xOPN_SW := TRUE; END_IF //for seamless transition   
    //Log
    fbLogger(sMsg:='Override expired', eSevr:=TcEventSeverity.Warning);
    
END_IF

//Override timer
tonOvrd(IN:=iq_stValve.pv_xOvrdOpn, PT:=tOvrd);

(* If Epics Command to close the Valve, check if PMPS and EPS are ok, otherwise Keep command set to open valve *)
IF NOT(iq_stValve.pv_xOPN_SW) AND ((NOT i_xPMPS_OK) OR (NOT i_xEPS_OK)) THEN
	//iq_stValve.pv_xOPN_SW := TRUE; // plc to only reset never to set this signal
END_IF
(* Reset the EPICS command to open the valve if the interlock is lost *) 
(* based on EPS ok state, EPS overrides OPN_OK*)
IF NOT iq_stValve.xOPN_OK THEN
	IF i_xEPS_OK THEN iq_stValve.pv_xOPN_SW := FALSE; iq_stValve.sErrorMessage := 'ILK Active';
	ELSE //iq_stValve.pv_xOPN_SW := TRUE;		// plc to only reset never to set this signal
	END_IF
END_IF

(* Here's where the valve opens *)
iq_stValve.q_xOPN_DO := (iq_stValve.pv_xOPN_SW AND iq_stValve.xOPN_OK) OR (tonOvrd.Q AND i_xOverrideMode);

(* When the valve  is open MPS is OK*)
xMPS_OK := (iq_stValve.eState=OPEN) OR (iq_stValve.eState=OPEN_F);//iq_stValve.i_xOpnLS; 

///Check valve moving postion timout
IF NOT iq_stValve.i_xClsLS AND tCLStimeout.Q THEN 
	iq_stValve.bErrorPresent := TRUE;
	iq_stValve.sErrorMessage := ' Close Timeout';
ELSIF NOT iq_stValve.i_xOpnLS AND tOPNtimeout.Q THEN 
	iq_stValve.bErrorPresent := TRUE; 
	iq_stValve.sErrorMessage := ' Open Timeout';
END_IF
IF (iq_stValve.eState=INVALID) THEN
	iq_stValve.bErrorPresent := TRUE; 
	iq_stValve.sErrorMessage := CONCAT(sPath,' Invalid Valve Position');
END_IF


(*Timers*)
tOPNtimeout(IN:= iq_stValve.q_xOPN_DO, PT := tTimeOutDuration );
tCLStimeout(IN:= NOT iq_stValve.q_xOPN_DO, PT := tTimeOutDuration);

// Log valve timeouts
tErrorPresent(CLK:=iq_stValve.bErrorPresent);
IF tErrorPresent.Q THEN fbLogger(sMsg:=iq_stValve.sErrorMessage, eSevr:=TcEventSeverity.Warning); END_IF

// Log valve open
tAction(CLK:= iq_stValve.q_xOPN_DO);
IF tAction.Q THEN fbLogger(sMsg:='Valve commanded open', eSevr:=TcEventSeverity.Info); END_IF

// Log override mode enabled
tOverrideActivated(CLK:= (tonOvrd.Q AND i_xOverrideMode));
IF tOverrideActivated.Q THEN fbLogger(sMsg:='Valve override mode activated', eSevr:=TcEventSeverity.Warning); END_IF

// Alarm reset
//////////////////////////////////////
ACT_ResetAlarms();

(*IO Mapping*)
ACT_IO();

(*FAST FAULT*)
fbFF(i_xOK := xMPS_OK,
    i_xReset := i_xReset,
	i_xAutoReset :=TRUE,
    io_fbFFHWO := io_fbFFHWO);

ACTION ACT_IO:
(*inputs*)
iq_stValve.i_xOpnLS := 	i_xOpnLS;
iq_stValve.i_xClsLS:=	i_xClsLS;
iq_stValve.xEXT_OK := i_xEXT_OK;
iq_stValve.xOverrideMode := i_xOverrideMode;
(*outputs*)
q_xOPN_DO:= iq_stValve.q_xOPN_DO;
q_xOPN_DO_2:= iq_stValve.q_xOPN_DO;


(*ILK Devices*)
iq_stValve.sIlkUSDeviceName := This^.i_stUSG.sPath;
iq_stValve.sIlkDSDeviceName := This^.i_stDSG.sPath;
END_ACTION

ACTION ACT_ResetAlarms:
iq_stValve.xERR_DifPres R= iq_stValve.pv_xAlmRst;
iq_stValve.xERR_SP R= iq_stValve.pv_xAlmRst;
iq_stValve.bErrorPresent R= iq_stValve.pv_xAlmRst;

IF ( iq_stValve.pv_xAlmRst) THEN
	iq_stValve.sErrorMessage :='';
END_IF
END_ACTION

METHOD PUBLIC M_IsClosed : BOOL
VAR_INPUT
END_VAR
M_IsClosed := (This^.iq_stValve.eState = E_ValvePositionState.CLOSED);
END_METHOD

METHOD PUBLIC M_IsOpen : BOOL
VAR_INPUT
END_VAR
M_IsOpen := (This^.iq_stValve.eState = E_ValvePositionState.OPEN);
END_METHOD

// Use this Methode to Open or close the valve by setting the OPN_SW to the input value.
METHOD PUBLIC M_Set_OPN_SW : BOOL
VAR_INPUT
		value:BOOL;
END_VAR
This^.iq_stValve.pv_xOPN_SW := value;
END_METHOD

END_FUNCTION_BLOCK

// POUs/Functions/Valves/FB_VGC
(* This function block implements basic functionality for Isolation Gate Valves*)
(* This function block interlock is as follows:
1. The valve can be opened when the difference between the pressures on both sides is
less than the maximum differential pressure.
2. This rule persists until the pressures on both sides are lower than the vacuum-setpoint.
3. Once at-vac, the valve will close if the pressure on either side rises above the setpoint.*)
(*This function block also implements PMPS and EPS interlocks, as well as Fast MPS trigger*)
{attribute 'no_check'}
{attribute 'reflection'} 
FUNCTION_BLOCK FB_VGC Extends FB_Valve
VAR_IN_OUT
	
END_VAR
VAR_INPUT
	(*Upstream Gauge, usually ion gauge*)
	i_stUSG	:	ST_VG;
	(*Downstream Gauge, usually ion gauge*)
	i_stDSG	:	ST_VG;
	{attribute 'pytmc' := '
    pv: Dis_DPIlk
	'}
	i_xDis_DPIlk : BOOL := FALSE;  (* Set to true when calling the function to disable the differential pressure interlock *)
	i_xPMPS_OK:	BOOL	; (*Set to True To switch off the bptm and PMPS Arbiter*)
	{attribute 'pytmc' := '
    pv: EPS_OK
	'}
	i_xEPS_OK:	BOOL	:= TRUE; (*External EPS interlock, Set to TRUE when no EPS interlock is required, otherwise set to correct interlock signal*)
	i_xExt_OK: BOOL; (*Other External Interlock, Set to True when no external interlock is required. If this Valve is neigboring a Fast Shutter this should be linked to the fast shutter xVAC_FAULT_OK*)
	i_xOverrideMode : BOOL; (*To be linked to global override bit. This Overrides Vacuum logic only, EPS, MPS and PMPS are still enforces*)
	// Reset fault
	{attribute 'pytmc' := '
    pv: FF_Reset
	'}
    i_xReset: BOOL;
	i_xIsAperture:BOOL :=FALSE; // Set tp True if this is an Aperture Valve, the MPS Fault will trip only when moving.
	i_sDevName : T_MaxString :=  'VGC'; // Device name for diagnostic
	i_nTransitionRootID: UDINT; //A unique transition Root ID that is equal to or greater than 1000
END_VAR
VAR_OUTPUT
	{attribute 'pytmc' := '
    pv:
	'}
	iq_stValve : ST_VGC; (* All valve data and states will be in this struct*)
	
	{attribute 'pytmc' := '
    pv: MPS_FAULT_OK
	field: ZNAM MPS FAULT ;
	field: ONAM MPS OK ;
	'}
	xMPS_OK:	BOOL; (*MPS Fast OK, is set when the Valve is Open*)
END_VAR
VAR_IN_OUT
	io_fbFFHWO    :    FB_HardwareFFOutput;
	fbArbiter: FB_Arbiter();
END_VAR
VAR
	// PMPS
	{attribute 'pytmc' := '
    pv: MPS_OK
	'}
	xPMPS_OK:	BOOL	; (*PMPS interlock*)
	bMoving : BOOL;
	bDone :BOOL;
	tBPTMtimeout:TON;
	bptm: BeamParameterTransitionManager;  
	FFO    :    FB_FastFault :=(
        i_DevName := 'VGC',
        i_Desc := 'Fault occurs when the valve is not in open state',
        i_TypeCode := 16#1010);
	//g_FastFaultOutput1	:	FB_HardwareFFOutput;	

	{attribute 'instance-path'}
	{attribute 'noinit'}
	sPath: STRING;
	
	rDiffPressAllowed	:	REAL := 22.5; // Torr, Default value comes from Vat Valve Manual
	rDiffPress : REAL;
	set : BOOL;
    reset: BOOL;
	  
	xFirstPass	:	BOOL;
	fbFSInit		:	R_TRIG;
	
	tonDelOK : TON;
	rtOK	:	R_TRIG;
	tonOvrd	:	TON;
	rtOpen	:	R_TRIG;
	ftClose: F_TRIG;
	
	tDelOK	:	TIME := T#60S;
	tOvrd	:	TIME := T#10s;
	
	
	(* Timeouts*)
	tTimeOutDuration: TIME:= T#30S;
	tOPNtimeout: TON;
	tCLStimeout:TON;
	
	
	(*IO*)
	i_xOpnLS	AT%I*: BOOL;
	i_xClsLS	AT%I*: BOOL;
	q_xOPN_DO	AT%Q*: BOOL;
    
    // For logging
    eVGCPrevState : E_VGC;
   
	
END_VAR

(* Vacuum gate valve
A. Wallace
16-10-29

A gate valve isolates vacuum volumes. Ideally it can be opened when a system is vented
to allow for faster pumping, and will close when high vacuum is lost.

The following behavior is good for valves in something like a gas attenuator.
This function block does the following:
1. The valve can be opened when the difference between the pressures on both sides is
less than the maximum differential pressure.
2. This rule persists until the pressures on both sides are lower than the vacuum-setpoint.
3. Once at-vac, the valve will close if the pressure on either side rises above the setpoint.

Alternatively, the differential pressure interlock can be disabled so the valve may only be opened
if the pressure on both sides is lower than the at-vacuum-setpoint. You want this behavior if 
the valve is to be used in a UHV section.

Hysteresis is employed to ensure a smooth transition from vented/pumping down, to at-vac.

Finally, an override system is built in so you can bypass all the interlocking logic and 
get back online.
*)
(* 10/1/2018 Margaret Ghaly included EPS, PMPS Checkes and MPS trigger signals*)


fbFSInit( CLK := TRUE, Q => xFirstPass);
(*IO Mapping*)
ACT_IO();

(* On first PLC pass, put valve into vented state, which implies a closed valve *)
IF xFirstPass THEN
	iq_stValve.eVGC_State := Vented;
	iq_stValve.pv_xOPN_SW := FALSE;
	FFO.i_DevName := i_sDevName;
END_IF


///Check valve position
IF iq_stValve.i_xClsLS AND  iq_stValve.i_xOpnLS THEN
	iq_stValve.eState:=INVALID;
ELSIF NOT iq_stValve.i_xClsLS AND iq_stValve.i_xOpnLS AND iq_stValve.q_xOPN_DO THEN 
	iq_stValve.eState:=OPEN;
ELSIF NOT iq_stValve.i_xClsLS AND iq_stValve.i_xOpnLS AND NOT iq_stValve.q_xOPN_DO THEN 
	iq_stValve.eState:=OPEN_F;
ELSIF iq_stValve.i_xClsLS AND NOT iq_stValve.i_xOpnLS AND NOT iq_stValve.q_xOPN_DO THEN 
	iq_stValve.eState:=CLOSED;
ELSIF NOT iq_stValve.i_xClsLS AND NOT iq_stValve.i_xOpnLS THEN 
	iq_stValve.eState:=MOVING;
ELSE
	iq_stValve.eState:=INVALID;
END_IF

// Update hysteresis
///////////////////////////////////////////////////
IF iq_stValve.rAT_VAC_SP_LAST <> iq_stValve.rAT_VAC_SP OR xFirstPass THEN
	iq_stValve.rAT_VAC_SP_LAST := iq_stValve.rAT_VAC_SP;
	iq_stValve.rAT_VAC_HYS := iq_stValve.rHYST_PERC * iq_stValve.rAT_VAC_SP;
END_IF

iq_stValve.rAT_VAC_HYS := LIMIT(0, iq_stValve.rAT_VAC_HYS, iq_stValve.rAT_VAC_SP);
IF iq_stValve.rAT_VAC_SP <> 0 THEN
	IF iq_stValve.rHYST_PERC <> (iq_stValve.rAT_VAC_HYS / iq_stValve.rAT_VAC_SP) THEN
		iq_stValve.rHYST_PERC := LIMIT(0, (iq_stValve.rAT_VAC_HYS / iq_stValve.rAT_VAC_SP) ,1);
	END_IF
END_IF
// Valve at vacuum check
///////////////////////////////////////////////////
	set := i_stUSG.rPRESS < iq_stValve.rAT_VAC_HYS AND i_stDSG.rPRESS < iq_stValve.rAT_VAC_HYS AND i_stUSG.xPRESS_OK AND i_stDSG.xPRESS_OK;
 	iq_stValve.xAT_VAC S= set;
	reset := i_stUSG.rPRESS > iq_stValve.rAT_VAC_SP OR i_stDSG.rPRESS > iq_stValve.rAT_VAC_SP OR NOT i_stUSG.xPRESS_OK OR NOT i_stDSG.xPRESS_OK;
	iq_stValve.xAT_VAC R= reset;
	
// Differential pressure check
///////////////////////////////////////////////////
	(* Calc the differential pressure across the valve *)
	rDiffPress := ABS(i_stUSG.rPRESS - i_stDSG.rPRESS);
	
	(* As long as the differential pressure is less than 30mbar, the valve is allowed to open *)
	IF rDiffPress <= rDiffPressAllowed AND i_stUSG.xPRESS_OK AND i_stDSG.xPRESS_OK THEN
		iq_stValve.xDP_OK := TRUE;
	ELSE
		iq_stValve.xDP_OK	:= FALSE;
		(* If the differential pressure is exceeded, even when the valve is open,
		the state is unexpected and triggers a fault, because it suggests that something
		is wrong with the valve, or gauges or mapping or there is a major leak on one side.*)
		iq_stValve.eVGC_State := ERR_DiffPress;
        iq_stValve.xERR_DifPres := TRUE;
	END_IF

// Valve state
///////////////////////////////////////////////////
CASE iq_stValve.eVGC_State OF
	Vented: (* The Vented state is used during pump down *)        
		(* Assuming the pump down went well, we are now at vacuum on both sides,
		so we move to the vacuum state, otherwise remain in the vented state *)
		IF iq_stValve.xAT_VAC AND (NOT (iq_stValve.xERR_DifPres)) AND (NOT (iq_stValve.xERR_SP)) AND (NOT (iq_stValve.xERR_ExtFault))THEN
		    iq_stValve.eVGC_State := AtVacuum;
		ELSE
		    iq_stValve.eVGC_State := Vented;
		END_IF
	
	AtVacuum:
		IF iq_stValve.xAT_VAC THEN
		(* If both pressure setpoints are made,
		then enable the differential pressure interlock, regardless of the valve state
		assuming we're using some kind of ion gauge where a pressure setpoint cannot be higher than 1E-4 T *)
		iq_stValve.eVGC_State := AtVacuum;
				
		ELSE
		
			(* If the valve is open (or in an unknown state) and either gauge is not at it's vacuum setpoint,
			we have a loss of vacuum error *)
			IF (iq_stValve.i_xOpnLS OR (NOT iq_stValve.i_xOpnLS AND NOT iq_stValve.i_xClsLS)) THEN
				iq_stValve.eVGC_State := ERR_LostVac;
				iq_stValve.xERR_SP := TRUE; //TAW changed this to the ERR_SP bool because I think that's what it was intended to be?
		
			(* Alternatively, if the valve is already closed and we lose pressure on one side,
			it was probably intentional venting, so we calmly move back to venting mode, and
			disable the differential pressure interlock *) //?? 
			ELSIF iq_stValve.i_xClsLS THEN
				iq_stValve.eVGC_State := Vented;
			END_IF
		
		END_IF
	
	ERR_DiffPress:       
		IF NOT (iq_stValve.xERR_DifPres) THEN
			IF iq_stValve.xAT_VAC AND (NOT (iq_stValve.xERR_DifPres)) AND (NOT (iq_stValve.xERR_SP)) AND (NOT (iq_stValve.xERR_ExtFault))THEN
		    	iq_stValve.eVGC_State := AtVacuum;
			ELSE
		    	iq_stValve.eVGC_State := Vented;
			END_IF
		END_IF
		
	
	ERR_LostVac:
		IF NOT (iq_stValve.xERR_SP) THEN
			IF iq_stValve.xAT_VAC AND (NOT (iq_stValve.xERR_DifPres)) AND (NOT (iq_stValve.xERR_SP)) AND (NOT (iq_stValve.xERR_ExtFault))THEN
		    	iq_stValve.eVGC_State := AtVacuum;
			ELSE
		    	iq_stValve.eVGC_State := Vented;
			END_IF
		END_IF
		
	ERR_ExtFault:
		IF NOT (iq_stValve.xERR_ExtFault) AND (i_xExt_OK) THEN
			IF iq_stValve.xAT_VAC AND (NOT (iq_stValve.xERR_DifPres)) AND (NOT (iq_stValve.xERR_SP)) AND (NOT (iq_stValve.xERR_ExtFault))THEN
		    	iq_stValve.eVGC_State := AtVacuum;
			ELSE
		    	iq_stValve.eVGC_State := Vented;
			END_IF
		END_IF
END_CASE

IF (NOT i_xExt_OK) AND (iq_stValve.eState=OPEN)  THEN
	iq_stValve.eVGC_State := ERR_ExtFault;
	iq_stValve.xERR_ExtFault := TRUE;
END_IF

// Interlock evaluation - with bypass for DP ILK bypass
///////////////////////////////////////////////
IF i_xDis_DPIlk THEN
	iq_stValve.xOPN_OK := iq_stValve.xEXT_OK; // AND iq_stValve.xDP_OK ;
ELSE
	iq_stValve.xOPN_OK := iq_stValve.xEXT_OK AND iq_stValve.xAT_VAC;
END_IF


(* Valve operation *)

(* Override logic *)
(* Goal: give ability to override, but do so in a way that people won't forget it.
Solution: Override only after ten seconds of override, protect against blips,
when the valve permission goes true for more than ten seconds consistently, remove override
*)

tonDelOK(IN:=iq_stValve.xOPN_OK, PT:=tDelOK);
rtOK(CLK:=tonDelOK.Q);
IF rtOK.Q AND iq_stValve.pv_xOvrdOpn THEN 
	iq_stValve.pv_xOvrdOpn :=FALSE;
	if (iq_stValve.eState = OPEN) AND (i_xOverrideMode) THEN iq_stValve.pv_xOPN_SW := TRUE; END_IF //for seamless transition   
    //Log
    fbLogger(sMsg:='Override expired', eSevr:=TcEventSeverity.Warning);
END_IF
// Release the Force Open bit when the system override is false
IF NOT (i_xOverrideMode) THEN  iq_stValve.pv_xOvrdOpn :=FALSE; END_IF
//Override timer
tonOvrd(IN:=iq_stValve.pv_xOvrdOpn, PT:=tOvrd);


(* Valve operation *)
(* Here's where we evaluate sw actions and operate the valve *)
(* Valve operation *)

ftClose(CLK:= iq_stValve.pv_xOPN_SW);
rtOpen(CLK:= iq_stValve.pv_xOPN_SW);


(*PMPS*)
IF NOT(i_xPMPS_OK) THEN
	ACT_PMPS();
END_IF
(*when interlock is lost the Valve closes regardless of the status of the PMPS and EPS*)
xPMPS_OK := i_xPMPS_OK OR (bptm.q_xTransitionAuthorized OR tBPTMtimeout.Q);
IF NOT (iq_stValve.xOPN_OK) THEN
	iq_stValve.pv_xOPN_SW:= FALSE; // Reset switch after inlk is lost
	iq_stValve.q_xOPN_DO := (iq_stValve.pv_xOPN_SW  AND iq_stValve.xOPN_OK) OR (tonOvrd.Q AND i_xOverrideMode);
ELSIF xPMPS_OK THEN 
	iq_stValve.q_xOPN_DO := (iq_stValve.pv_xOPN_SW  AND iq_stValve.xOPN_OK) OR (tonOvrd.Q AND i_xOverrideMode);
//ELSIF NOT (i_xPMPS_OK) THEN
	// Only override mode
	//iq_stValve.q_xOPN_DO := (tonOvrd.Q AND i_xOverrideMode);
END_IF


(*MPS Fault setting*)
If (i_xIsAperture ) THEN 
	(* When the valve  is open or in Closed position MPS is OK, Fault while moving*)
	xMPS_OK := (i_xOpnLS  AND q_xOPN_DO) XOR (i_xClsLS  AND NOT q_xOPN_DO); 
ELSE
	(* When the valve  is open MPS is OK*)
	xMPS_OK := i_xOpnLS AND NOT i_xClsLS AND q_xOPN_DO; 
END_IF


///Check valve moving postion timout
IF NOT iq_stValve.i_xClsLS AND tCLStimeout.Q THEN 
	iq_stValve.bErrorPresent := TRUE;
	iq_stValve.sErrorMessage := 'Close Timeout';
ELSIF NOT iq_stValve.i_xOpnLS AND tOPNtimeout.Q THEN 
	iq_stValve.bErrorPresent := TRUE; 
	iq_stValve.sErrorMessage := 'Open Timeout';
END_IF
IF (iq_stValve.eState=INVALID) THEN
	iq_stValve.bErrorPresent := TRUE; 
	iq_stValve.sErrorMessage := CONCAT(sPath,'Invalid Valve Position');
END_IF


(*Timers*)
tOPNtimeout(IN:= iq_stValve.q_xOPN_DO, PT := tTimeOutDuration );
tCLStimeout(IN:= NOT iq_stValve.q_xOPN_DO, PT := tTimeOutDuration);


// Alarm reset
//////////////////////////////////////
ACT_ResetAlarms();

(*IO Mapping*)
ACT_IO();

// Log States and triggers
ACT_Logger();



(*FAST FAULT*)
FFO(i_xOK := xMPS_OK,
    i_xReset := i_xReset,
	i_xAutoReset :=TRUE,
    io_fbFFHWO := io_fbFFHWO);

ACTION ACT_IO:
(*inputs*)
iq_stValve.i_xOpnLS := 	i_xOpnLS;
iq_stValve.i_xClsLS:=	i_xClsLS;
iq_stValve.xEXT_OK := i_xEXT_OK;
iq_stValve.xOverrideMode := i_xOverrideMode;
(*outputs*)
q_xOPN_DO:= iq_stValve.q_xOPN_DO;

(*ILK Devices*)
iq_stValve.sIlkUSDeviceName := This^.i_stUSG.sPath;
iq_stValve.sIlkDSDeviceName := This^.i_stDSG.sPath;
END_ACTION

ACTION ACT_Logger:
// ILK logger

IF NOT (iq_stValve.xOPN_OK) AND (ePrevState = OPEN) AND NOT (TonOvrd.Q) THEN
 		fbLogger(sMsg:='Lost interlock ok bit while valve was open.', eSevr:=TcEventSeverity.Critical);  	
END_IF


//Positiong STATE Logger  
IF ePrevState <> iq_stValve.eState THEN
	  CASE iq_stValve.eState OF
		INVALID:
			fbLogger(sMsg:='Valve invalid position.', eSevr:=TcEventSeverity.Critical);
  		MOVING:
			fbLogger(sMsg:='Valve moving', eSevr:=TcEventSeverity.Warning);
		OPEN:
			fbLogger(sMsg:='Valve Open.', eSevr:=TcEventSeverity.Info);
		OPEN_F:
			fbLogger(sMsg:='Valve Open.', eSevr:=TcEventSeverity.Info);
		CLOSED:
			fbLogger(sMsg:='Valve closed.', eSevr:=TcEventSeverity.Info);
	  END_CASE
	  ePrevState := iq_stValve.eState;  
  END_IF
 
 //Pressure STATE Logger  
IF eVGCPrevState <> iq_stValve.eVGC_State THEN
	  CASE iq_stValve.eVGC_State OF
		Vented:
			 fbLogger(sMsg:='Vented', eSevr:=TcEventSeverity.Info);
  		AtVacuum:
			 fbLogger(sMsg:='Vacuum setpoint satisfied', eSevr:=TcEventSeverity.Info);
		ERR_DiffPress:
			 fbLogger(sMsg:='Potential accidental vent.', eSevr:=TcEventSeverity.Critical);
		ERR_LostVac:
			fbLogger(sMsg:='Unexpected loss of vacuum while valve was open or moving.', eSevr:=TcEventSeverity.Critical);
		ERR_ExtFault:
			 fbLogger(sMsg:='Lost external interlock while valve was open.', eSevr:=TcEventSeverity.Critical);
	  END_CASE
	  eVGCPrevState := iq_stValve.eVGC_State;  
  END_IF
  


// Log valve timeouts
tErrorPresent(CLK:=iq_stValve.bErrorPresent);
IF tErrorPresent.Q THEN fbLogger(sMsg:=iq_stValve.sErrorMessage, eSevr:=TcEventSeverity.Warning); END_IF

// Log valve open
tAction(CLK:= iq_stValve.q_xOPN_DO);
IF tAction.Q THEN fbLogger(sMsg:='Valve commanded open', eSevr:=TcEventSeverity.Info); END_IF

// Log override mode enabled
tOverrideActivated(CLK:= (tonOvrd.Q AND i_xOverrideMode));
IF tOverrideActivated.Q THEN fbLogger(sMsg:='Valve override mode activated', eSevr:=TcEventSeverity.Warning); END_IF
END_ACTION

